C08989=1033.832,386.586,-137.871,173.247,46.071,159.158
C08990=1033.841,386.832,-137.913,173.256,46.074,159.159
C08991=1033.850,387.077,-137.956,173.264,46.078,159.161
C08992=1033.859,387.324,-137.998,173.272,46.082,159.163
C08993=1033.868,387.571,-138.041,173.280,46.085,159.165
C08994=1033.878,387.816,-138.083,173.289,46.089,159.167
C08995=1033.886,388.062,-138.126,173.297,46.092,159.169
C08996=1033.895,388.309,-138.168,173.306,46.096,159.171
C08997=1033.904,388.554,-138.210,173.314,46.100,159.173
C08998=1033.913,388.801,-138.254,173.324,46.103,159.175
C08999=1033.923,389.047,-138.296,173.332,46.106,159.176
C09000=1033.931,389.293,-138.339,173.341,46.110,159.178
C09001=1033.941,389.539,-138.382,173.350,46.114,159.180
C09002=1033.950,389.785,-138.424,173.358,46.117,159.182
C09003=1033.959,390.031,-138.467,173.367,46.121,159.184
C09004=1033.969,390.278,-138.510,173.376,46.125,159.186
C09005=1033.977,390.524,-138.553,173.384,46.129,159.188
C09006=1033.987,390.770,-138.597,173.393,46.132,159.190
C09007=1033.996,391.016,-138.640,173.402,46.136,159.192
C09008=1034.005,391.261,-138.682,173.410,46.140,159.194
C09009=1034.014,391.508,-138.726,173.420,46.143,159.196
C09010=1034.024,391.753,-138.769,173.429,46.147,159.198
C09011=1034.033,392.000,-138.812,173.437,46.151,159.200
C09012=1034.042,392.246,-138.855,173.446,46.155,159.202
C09013=1034.051,392.492,-138.899,173.455,46.159,159.204
C09014=1034.060,392.726,-138.940,173.463,46.162,159.206
C09015=1034.069,392.960,-138.981,173.472,46.166,159.208
C09016=1034.078,393.195,-139.022,173.481,46.170,159.210
C09017=1034.087,393.430,-139.063,173.489,46.173,159.212
C09018=1034.096,393.664,-139.105,173.498,46.177,159.214
C09019=1034.105,393.898,-139.146,173.507,46.181,159.216
C09020=1034.114,394.134,-139.188,173.515,46.184,159.218
C09021=1034.123,394.368,-139.229,173.524,46.188,159.220
C09022=1034.132,394.614,-139.273,173.533,46.192,159.222
C09023=1034.141,394.860,-139.317,173.542,46.196,159.224
C09024=1034.151,395.105,-139.360,173.551,46.200,159.226
C09025=1034.160,395.352,-139.404,173.560,46.204,159.228
C09026=1034.170,395.598,-139.448,173.570,46.208,159.230
C09027=1034.179,395.843,-139.491,173.579,46.212,159.232
C09028=1034.188,396.089,-139.535,173.588,46.216,159.234
C09029=1034.198,396.335,-139.579,173.598,46.220,159.237
C09030=1034.207,396.582,-139.623,173.607,46.224,159.239
C09031=1034.217,396.827,-139.667,173.617,46.228,159.241
C09032=1034.227,397.072,-139.711,173.626,46.233,159.243
C09033=1034.236,397.318,-139.755,173.635,46.237,159.245
C09034=1034.245,397.565,-139.799,173.645,46.241,159.247
C09035=1034.256,397.810,-139.843,173.654,46.245,159.250
C09036=1034.265,398.056,-139.887,173.664,46.249,159.252
C09037=1034.275,398.302,-139.932,173.673,46.253,159.254
C09038=1034.284,398.548,-139.976,173.683,46.257,159.256
C09039=1034.294,398.794,-140.019,173.692,46.261,159.258
C09040=1034.304,399.039,-140.064,173.701,46.265,159.260
C09041=1034.313,399.286,-140.108,173.712,46.270,159.263
C09042=1034.323,399.532,-140.152,173.721,46.274,159.265
C09043=1034.332,399.777,-140.197,173.731,46.278,159.267
C09044=1034.343,400.022,-140.241,173.740,46.283,159.270
C09045=1034.352,400.269,-140.286,173.750,46.287,159.272
C09046=1034.362,400.514,-140.330,173.759,46.292,159.274
C09047=1034.371,400.760,-140.375,173.769,46.296,159.276
C09048=1034.381,401.006,-140.419,173.779,46.300,159.279
C09049=1034.391,401.251,-140.464,173.788,46.304,159.281
C09050=1034.401,401.497,-140.509,173.799,46.309,159.283
C09051=1034.410,401.742,-140.554,173.809,46.313,159.286
C09052=1034.420,401.989,-140.598,173.818,46.317,159.288
C09053=1034.430,402.235,-140.643,173.828,46.322,159.290
C09054=1034.440,402.480,-140.688,173.838,46.326,159.293
C09055=1034.449,402.726,-140.733,173.848,46.331,159.295
C09056=1034.460,402.972,-140.778,173.858,46.336,159.297
C09057=1034.470,403.217,-140.823,173.868,46.340,159.300
C09058=1034.478,403.463,-140.868,173.879,46.345,159.302
C09059=1034.489,403.708,-140.914,173.888,46.349,159.305
C09060=1034.499,403.954,-140.959,173.898,46.354,159.307
C09061=1034.509,404.200,-141.004,173.908,46.358,159.309
C09062=1034.518,404.445,-141.049,173.919,46.363,159.312
C09063=1034.529,404.691,-141.094,173.929,46.367,159.314
C09064=1034.538,404.937,-141.140,173.939,46.372,159.317
C09065=1034.548,405.183,-141.185,173.949,46.377,159.319
C09066=1034.558,405.428,-141.231,173.959,46.382,159.322
C09067=1034.569,405.674,-141.276,173.970,46.386,159.324
C09068=1034.579,405.919,-141.321,173.980,46.390,159.326
C09069=1034.588,406.166,-141.367,173.990,46.396,159.329
C09070=1034.598,406.403,-141.412,174.001,46.400,159.331
C09071=1034.608,406.640,-141.455,174.010,46.405,159.334
C09072=1034.618,406.877,-141.499,174.020,46.409,159.336
C09073=1034.627,407.114,-141.543,174.031,46.414,159.339
C09074=1034.637,407.355,-141.588,174.041,46.419,159.341
C09075=1034.647,407.596,-141.633,174.052,46.423,159.344
C09076=1034.658,407.837,-141.678,174.062,46.427,159.346
C09077=1034.667,408.077,-141.722,174.071,46.433,159.349
C09078=1034.677,408.318,-141.767,174.082,46.437,159.351
C09079=1034.688,408.558,-141.813,174.092,46.442,159.354
C09080=1034.698,408.799,-141.857,174.103,46.447,159.356
C09081=1034.707,409.040,-141.903,174.113,46.452,159.359
C09082=1034.718,409.286,-141.949,174.124,46.457,159.361
C09083=1034.728,409.531,-141.994,174.135,46.461,159.364
C09084=1034.739,409.776,-142.040,174.146,46.466,159.367
C09085=1034.749,410.022,-142.086,174.157,46.471,159.369
C09086=1034.760,410.267,-142.133,174.167,46.476,159.372
C09087=1034.770,410.513,-142.179,174.178,46.481,159.374
C09088=1034.781,410.758,-142.225,174.190,46.486,159.377
C09089=1034.791,411.004,-142.271,174.201,46.491,159.380
C09090=1034.802,411.249,-142.318,174.211,46.496,159.382
C09091=1034.812,411.495,-142.364,174.222,46.501,159.385
C09092=1034.822,411.740,-142.411,174.234,46.507,159.388
C09093=1034.833,411.986,-142.457,174.244,46.512,159.391
C09094=1034.843,412.231,-142.504,174.255,46.517,159.393
C09095=1034.854,412.477,-142.550,174.267,46.522,159.396
C09096=1034.864,412.722,-142.597,174.278,46.527,159.399
C09097=1034.874,412.967,-142.645,174.289,46.533,159.402
C09098=1034.885,413.213,-142.691,174.300,46.537,159.404
C09099=1034.895,413.458,-142.738,174.311,46.543,159.407
C09100=1034.906,413.703,-142.784,174.323,46.548,159.410
C09101=1034.917,413.949,-142.832,174.334,46.554,159.413
C09102=1034.928,414.194,-142.879,174.346,46.558,159.416
C09103=1034.938,414.439,-142.926,174.357,46.564,159.418
C09104=1034.949,414.684,-142.972,174.369,46.569,159.421
C09105=1034.959,414.930,-143.020,174.380,46.574,159.424
C09106=1034.970,415.176,-143.067,174.392,46.580,159.427
C09107=1034.981,415.420,-143.114,174.403,46.585,159.430
C09108=1034.991,415.666,-143.161,174.415,46.591,159.433
C09109=1035.002,415.911,-143.208,174.426,46.596,159.436
C09110=1035.013,416.157,-143.255,174.438,46.602,159.439
C09111=1035.025,416.402,-143.303,174.450,46.607,159.441
C09112=1035.035,416.647,-143.350,174.461,46.613,159.444
C09113=1035.046,416.893,-143.397,174.473,46.618,159.447
C09114=1035.057,417.137,-143.445,174.485,46.623,159.450
C09115=1035.068,417.383,-143.493,174.497,46.629,159.453
C09116=1035.078,417.628,-143.541,174.509,46.635,159.456
C09117=1035.090,417.874,-143.588,174.521,46.640,159.459
C09118=1035.100,418.118,-143.636,174.533,46.646,159.462
C09119=1035.111,418.364,-143.684,174.545,46.651,159.465
C09120=1035.121,418.609,-143.731,174.556,46.657,159.468
C09121=1035.132,418.854,-143.779,174.568,46.663,159.471
C09122=1035.144,419.100,-143.828,174.581,46.668,159.474
C09123=1035.155,419.344,-143.875,174.593,46.674,159.477
C09124=1035.166,419.589,-143.923,174.605,46.680,159.480
C09125=1035.177,419.835,-143.972,174.618,46.685,159.484
C09126=1035.187,420.079,-144.020,174.630,46.691,159.487
C09127=1035.199,420.325,-144.068,174.642,46.697,159.490
C09128=1035.210,420.570,-144.116,174.655,46.703,159.493
C09129=1035.222,420.815,-144.164,174.667,46.709,159.496
C09130=1035.233,421.061,-144.212,174.679,46.714,159.499
C09131=1035.243,421.305,-144.260,174.692,46.720,159.502
C09132=1035.255,421.550,-144.309,174.704,46.726,159.506
C09133=1035.266,421.795,-144.357,174.717,46.732,159.509
C09134=1035.277,422.041,-144.406,174.729,46.738,159.512
C09135=1035.288,422.286,-144.455,174.742,46.744,159.515
C09136=1035.300,422.531,-144.502,174.754,46.750,159.518
C09137=1035.311,422.775,-144.551,174.767,46.756,159.522
C09138=1035.323,423.021,-144.600,174.780,46.762,159.525
C09139=1035.334,423.266,-144.649,174.793,46.768,159.528
C09140=1035.346,423.511,-144.697,174.805,46.774,159.531
C09141=1035.357,423.756,-144.746,174.818,46.780,159.535
C09142=1035.368,424.001,-144.795,174.832,46.786,159.538
C09143=1035.380,424.246,-144.844,174.844,46.792,159.541
C09144=1035.391,424.490,-144.893,174.857,46.798,159.545
C09145=1035.403,424.735,-144.942,174.871,46.804,159.548
C09146=1035.414,424.982,-144.992,174.883,46.810,159.551
C09147=1035.425,425.226,-145.041,174.896,46.817,159.555
C09148=1035.437,425.470,-145.090,174.910,46.823,159.558
C09149=1035.448,425.715,-145.139,174.923,46.829,159.561
C09150=1035.460,425.961,-145.189,174.936,46.835,159.565
C09151=1035.471,426.205,-145.238,174.949,46.842,159.568
C09152=1035.483,426.450,-145.287,174.963,46.848,159.572
C09153=1035.495,426.695,-145.337,174.976,46.854,159.575
C09154=1035.507,426.940,-145.386,174.990,46.861,159.579
C09155=1035.519,427.185,-145.435,175.003,46.867,159.582
C09156=1035.530,427.429,-145.485,175.016,46.873,159.585
C09157=1035.542,427.675,-145.535,175.030,46.879,159.589
C09158=1035.553,427.919,-145.585,175.043,46.886,159.593
C09159=1035.566,428.164,-145.635,175.057,46.892,159.596
C09160=1035.577,428.408,-145.685,175.071,46.899,159.600
C09161=1035.589,428.654,-145.735,175.084,46.905,159.603
C09162=1035.600,428.898,-145.784,175.099,46.912,159.607
C09163=1035.612,429.143,-145.835,175.113,46.919,159.610
C09164=1035.624,429.387,-145.885,175.127,46.925,159.614
C09165=1035.636,429.632,-145.935,175.141,46.931,159.618
C09166=1035.647,429.877,-145.986,175.154,46.939,159.621
C09167=1035.659,430.121,-146.035,175.168,46.945,159.625
C09168=1035.672,430.366,-146.085,175.182,46.952,159.629
C09169=1035.683,430.611,-146.137,175.196,46.958,159.632
C09170=1035.696,430.855,-146.187,175.211,46.965,159.636
C09171=1035.708,431.100,-146.237,175.225,46.972,159.640
C09172=1035.719,431.345,-146.287,175.239,46.979,159.644
C09173=1035.732,431.589,-146.338,175.254,46.985,159.647
C09174=1035.744,431.834,-146.388,175.268,46.992,159.651
C09175=1035.757,432.078,-146.439,175.282,46.999,159.655
C09176=1035.768,432.323,-146.490,175.297,47.005,159.659
C09177=1035.781,432.567,-146.541,175.312,47.012,159.663
C09178=1035.793,432.811,-146.591,175.326,47.019,159.666
C09179=1035.805,433.057,-146.642,175.341,47.026,159.670
C09180=1035.818,433.301,-146.693,175.355,47.033,159.674
C09181=1035.830,433.545,-146.744,175.371,47.040,159.678
C09182=1035.842,433.789,-146.795,175.385,47.047,159.682
C09183=1035.855,434.034,-146.846,175.400,47.054,159.686
C09184=1035.867,434.279,-146.898,175.415,47.060,159.690
C09185=1035.880,434.523,-146.948,175.430,47.068,159.694
C09186=1035.893,434.768,-147.000,175.445,47.074,159.697
C09187=1035.905,435.013,-147.051,175.460,47.082,159.701
C09188=1035.917,435.257,-147.102,175.475,47.089,159.705
C09189=1035.930,435.501,-147.154,175.490,47.096,159.709
C09190=1035.942,435.746,-147.206,175.505,47.103,159.713
C09191=1035.955,435.990,-147.257,175.521,47.110,159.717
C09192=1035.967,436.234,-147.309,175.537,47.117,159.721
C09193=1035.980,436.479,-147.360,175.552,47.125,159.726
C09194=1035.993,436.725,-147.412,175.567,47.132,159.730
C09195=1036.006,436.971,-147.465,175.583,47.139,159.734
C09196=1036.018,437.216,-147.516,175.598,47.147,159.738
C09197=1036.031,437.462,-147.569,175.614,47.154,159.742
C09198=1036.044,437.707,-147.621,175.630,47.161,159.746
C09199=1036.057,437.951,-147.674,175.646,47.169,159.751
C09200=1036.070,438.195,-147.725,175.662,47.176,159.755
C09201=1036.082,438.440,-147.778,175.677,47.184,159.759
C09202=1036.095,438.683,-147.830,175.693,47.191,159.763
C09203=1036.108,438.928,-147.882,175.709,47.198,159.767
C09204=1036.121,439.172,-147.934,175.725,47.206,159.772
C09205=1036.134,439.417,-147.987,175.741,47.214,159.776
C09206=1036.147,439.660,-148.039,175.757,47.221,159.780
C09207=1036.160,439.904,-148.091,175.773,47.228,159.785
C09208=1036.173,440.148,-148.145,175.789,47.236,159.789
C09209=1036.186,440.393,-148.196,175.807,47.243,159.793
C09210=1036.199,440.637,-148.250,175.823,47.251,159.798
C09211=1036.212,440.881,-148.302,175.839,47.259,159.802
C09212=1036.225,441.125,-148.355,175.856,47.267,159.807
C09213=1036.238,441.369,-148.408,175.872,47.274,159.811
C09214=1036.252,441.613,-148.461,175.889,47.282,159.816
C09215=1036.265,441.857,-148.514,175.906,47.290,159.820
C09216=1036.278,442.101,-148.568,175.922,47.297,159.825
C09217=1036.292,442.345,-148.621,175.940,47.305,159.829
C09218=1036.305,442.588,-148.673,175.956,47.313,159.834
C09219=1036.319,442.832,-148.727,175.973,47.320,159.838
C09220=1036.332,443.076,-148.780,175.990,47.329,159.843
C09221=1036.345,443.320,-148.833,176.008,47.336,159.847
C09222=1036.359,443.563,-148.886,176.024,47.344,159.852
C09223=1036.372,443.807,-148.939,176.042,47.352,159.857
C09224=1036.386,444.050,-148.993,176.058,47.360,159.861
C09225=1036.399,444.294,-149.046,176.076,47.368,159.866
C09226=1036.414,444.537,-149.099,176.094,47.376,159.870
C09227=1036.429,444.780,-149.150,176.111,47.384,159.875
C09228=1036.445,445.024,-149.203,176.129,47.391,159.880
C09229=1036.461,445.267,-149.254,176.146,47.399,159.884
C09230=1036.478,445.511,-149.305,176.164,47.406,159.889
C09231=1036.495,445.755,-149.355,176.182,47.413,159.893
C09232=1036.513,445.999,-149.405,176.200,47.421,159.898
C09233=1036.531,446.243,-149.455,176.218,47.428,159.903
C09234=1036.550,446.486,-149.503,176.236,47.435,159.907
C09235=1036.569,446.731,-149.553,176.254,47.442,159.911
C09236=1036.589,446.975,-149.601,176.272,47.449,159.916
C09237=1036.609,447.220,-149.649,176.291,47.456,159.921
C09238=1036.630,447.464,-149.696,176.309,47.462,159.925
C09239=1036.652,447.708,-149.743,176.327,47.469,159.929
C09240=1036.673,447.953,-149.789,176.346,47.475,159.934
C09241=1036.697,448.198,-149.835,176.364,47.482,159.938
C09242=1036.719,448.442,-149.881,176.383,47.488,159.943
C09243=1036.743,448.687,-149.926,176.401,47.495,159.947
C09244=1036.767,448.931,-149.971,176.421,47.501,159.952
C09245=1036.792,449.177,-150.015,176.440,47.507,159.956
C09246=1036.817,449.422,-150.059,176.459,47.513,159.961
C09247=1036.843,449.667,-150.102,176.478,47.519,159.965
C09248=1036.869,449.912,-150.145,176.497,47.525,159.969
C09249=1036.896,450.157,-150.188,176.517,47.530,159.974
C09250=1036.924,450.403,-150.229,176.536,47.536,159.978
C09251=1036.951,450.649,-150.271,176.555,47.541,159.982
C09252=1036.980,450.893,-150.313,176.575,47.548,159.987
C09253=1037.009,451.139,-150.353,176.594,47.553,159.991
C09254=1037.046,451.441,-150.403,176.619,47.560,159.996
C09255=1037.083,451.744,-150.451,176.644,47.566,160.002
C09256=1037.122,452.046,-150.499,176.668,47.572,160.007
C09257=1037.160,452.347,-150.547,176.693,47.578,160.012
C09258=1036.869,452.403,-150.871,176.696,47.649,160.034
C09259=1036.832,452.115,-150.826,176.672,47.644,160.029
C09260=1036.796,451.826,-150.779,176.648,47.637,160.024
C09261=1036.760,451.537,-150.733,176.625,47.632,160.019
C09262=1036.724,451.248,-150.686,176.602,47.626,160.014
C09263=1036.695,451.003,-150.646,176.582,47.620,160.010
C09264=1036.666,450.758,-150.605,176.562,47.615,160.006
C09265=1036.638,450.512,-150.564,176.543,47.609,160.001
C09266=1036.610,450.266,-150.522,176.523,47.604,159.997
C09267=1036.583,450.021,-150.480,176.504,47.598,159.992
C09268=1036.557,449.776,-150.437,176.484,47.592,159.988
C09269=1036.531,449.531,-150.394,176.465,47.586,159.984
C09270=1036.504,449.286,-150.350,176.446,47.580,159.979
C09271=1036.480,449.041,-150.307,176.427,47.574,159.975
C09272=1036.455,448.796,-150.261,176.408,47.569,159.971
C09273=1036.431,448.551,-150.217,176.389,47.562,159.966
C09274=1036.407,448.306,-150.171,176.371,47.556,159.962
C09275=1036.385,448.062,-150.126,176.351,47.549,159.957
C09276=1036.363,447.816,-150.080,176.333,47.543,159.953
C09277=1036.341,447.572,-150.033,176.314,47.537,159.948
C09278=1036.319,447.328,-149.986,176.296,47.530,159.944
C09279=1036.298,447.084,-149.938,176.278,47.523,159.939
C09280=1036.279,446.839,-149.890,176.259,47.517,159.935
C09281=1036.259,446.595,-149.841,176.241,47.510,159.930
C09282=1036.240,446.351,-149.794,176.223,47.503,159.926
C09283=1036.221,446.107,-149.744,176.204,47.496,159.921
C09284=1036.203,445.863,-149.694,176.187,47.489,159.917
C09285=1036.185,445.619,-149.644,176.168,47.482,159.912
C09286=1036.169,445.375,-149.593,176.151,47.474,159.908
C09287=1036.152,445.132,-149.542,176.133,47.467,159.903
C09288=1036.137,444.888,-149.491,176.116,47.459,159.898
C09289=1036.121,444.645,-149.439,176.098,47.452,159.894
C09290=1036.106,444.402,-149.387,176.081,47.444,159.889
C09291=1036.092,444.159,-149.333,176.063,47.437,159.885
C09292=1036.078,443.915,-149.281,176.046,47.429,159.880
C09293=1036.065,443.672,-149.227,176.029,47.421,159.875
C09294=1036.051,443.429,-149.173,176.011,47.413,159.871
C09295=1036.038,443.185,-149.120,175.994,47.405,159.866
C09296=1036.025,442.941,-149.067,175.977,47.398,159.862
C09297=1036.011,442.697,-149.014,175.960,47.390,159.857
C09298=1035.997,442.453,-148.961,175.943,47.382,159.852
C09299=1035.984,442.209,-148.907,175.926,47.375,159.848
C09300=1035.970,441.966,-148.854,175.910,47.367,159.843
C09301=1035.957,441.721,-148.802,175.892,47.359,159.839
C09302=1035.944,441.477,-148.749,175.876,47.351,159.834
C09303=1035.931,441.233,-148.695,175.859,47.344,159.830
C09304=1035.917,440.989,-148.643,175.842,47.336,159.825
C09305=1035.904,440.745,-148.590,175.826,47.328,159.821
C09306=1035.891,440.501,-148.537,175.809,47.321,159.817
C09307=1035.878,440.257,-148.484,175.793,47.314,159.812
C09308=1035.866,440.013,-148.432,175.777,47.306,159.808
C09309=1035.852,439.769,-148.379,175.761,47.298,159.804
C09310=1035.839,439.525,-148.327,175.744,47.291,159.799
C09311=1035.826,439.281,-148.273,175.728,47.284,159.795
C09312=1035.813,439.036,-148.222,175.711,47.276,159.791
C09313=1035.800,438.793,-148.169,175.695,47.269,159.786
C09314=1035.787,438.548,-148.118,175.679,47.262,159.782
C09315=1035.774,438.304,-148.065,175.664,47.255,159.778
C09316=1035.762,438.060,-148.013,175.648,47.247,159.774
C09317=1035.748,437.815,-147.961,175.632,47.239,159.769
C09318=1035.736,437.571,-147.909,175.617,47.233,159.765
C09319=1035.723,437.324,-147.855,175.600,47.225,159.761
C09320=1035.710,437.076,-147.803,175.584,47.218,159.757
C09321=1035.697,436.829,-147.751,175.569,47.211,159.753
C09322=1035.684,436.582,-147.698,175.553,47.203,159.749
C09323=1035.672,436.338,-147.647,175.538,47.196,159.745
C09324=1035.659,436.094,-147.595,175.522,47.189,159.740
C09325=1035.646,435.849,-147.543,175.506,47.182,159.736
C09326=1035.634,435.605,-147.492,175.492,47.175,159.732
C09327=1035.622,435.361,-147.441,175.476,47.168,159.728
C09328=1035.608,435.116,-147.389,175.461,47.161,159.724
C09329=1035.596,434.872,-147.337,175.446,47.154,159.720
C09330=1035.584,434.628,-147.286,175.431,47.147,159.716
C09331=1035.572,434.383,-147.235,175.415,47.140,159.712
C09332=1035.559,434.138,-147.184,175.401,47.133,159.709
C09333=1035.547,433.894,-147.132,175.387,47.126,159.705
C09334=1035.534,433.650,-147.082,175.371,47.119,159.701
C09335=1035.522,433.405,-147.032,175.356,47.112,159.697
C09336=1035.510,433.160,-146.980,175.341,47.106,159.693
C09337=1035.497,432.915,-146.929,175.326,47.099,159.689
C09338=1035.484,432.671,-146.878,175.312,47.092,159.685
C09339=1035.472,432.426,-146.827,175.298,47.085,159.681
C09340=1035.460,432.182,-146.777,175.283,47.078,159.678
C09341=1035.447,431.938,-146.726,175.268,47.072,159.674
C09342=1035.435,431.694,-146.676,175.254,47.065,159.670
C09343=1035.424,431.448,-146.625,175.239,47.059,159.666
C09344=1035.411,431.204,-146.575,175.225,47.052,159.663
C09345=1035.399,430.959,-146.524,175.211,47.045,159.659
C09346=1035.387,430.714,-146.474,175.197,47.039,159.655
C09347=1035.375,430.470,-146.423,175.182,47.032,159.651
C09348=1035.363,430.226,-146.373,175.168,47.025,159.648
C09349=1035.351,429.981,-146.323,175.154,47.019,159.644
C09350=1035.339,429.736,-146.272,175.140,47.012,159.641
C09351=1035.327,429.491,-146.222,175.126,47.006,159.637
C09352=1035.316,429.247,-146.172,175.112,47.000,159.633
C09353=1035.304,429.002,-146.122,175.098,46.992,159.630
C09354=1035.292,428.758,-146.072,175.084,46.986,159.626
C09355=1035.280,428.513,-146.022,175.070,46.980,159.622
C09356=1035.269,428.268,-145.972,175.056,46.973,159.619
C09357=1035.257,428.023,-145.922,175.042,46.967,159.615
C09358=1035.245,427.779,-145.873,175.029,46.960,159.612
C09359=1035.233,427.534,-145.822,175.016,46.955,159.608
C09360=1035.222,427.289,-145.773,175.002,46.948,159.605
C09361=1035.210,427.044,-145.723,174.989,46.942,159.601
C09362=1035.198,426.799,-145.674,174.975,46.936,159.598
C09363=1035.186,426.554,-145.625,174.961,46.929,159.594
C09364=1035.174,426.310,-145.575,174.948,46.923,159.591
C09365=1035.162,426.064,-145.525,174.934,46.917,159.587
C09366=1035.151,425.820,-145.476,174.921,46.911,159.584
C09367=1035.140,425.575,-145.427,174.907,46.904,159.581
C09368=1035.128,425.329,-145.377,174.895,46.898,159.577
C09369=1035.117,425.085,-145.328,174.881,46.892,159.574
C09370=1035.105,424.840,-145.279,174.868,46.886,159.571
C09371=1035.094,424.596,-145.230,174.856,46.880,159.567
C09372=1035.083,424.350,-145.181,174.842,46.874,159.564
C09373=1035.071,424.105,-145.132,174.829,46.868,159.561
C09374=1035.059,423.860,-145.083,174.816,46.862,159.557
C09375=1035.048,423.615,-145.034,174.803,46.856,159.554
C09376=1035.037,423.371,-144.985,174.790,46.850,159.551
C09377=1035.025,423.125,-144.937,174.778,46.844,159.548
C09378=1035.014,422.880,-144.888,174.764,46.838,159.544
C09379=1035.003,422.633,-144.839,174.752,46.832,159.541
C09380=1034.990,422.386,-144.790,174.739,46.826,159.538
C09381=1034.979,422.138,-144.741,174.726,46.821,159.534
C09382=1034.968,421.890,-144.692,174.713,46.814,159.531
C09383=1034.957,421.645,-144.644,174.701,46.809,159.528
C09384=1034.945,421.400,-144.595,174.688,46.803,159.525
C09385=1034.934,421.155,-144.547,174.676,46.797,159.522
C09386=1034.923,420.910,-144.499,174.663,46.791,159.519
C09387=1034.912,420.665,-144.451,174.651,46.786,159.515
C09388=1034.901,420.421,-144.402,174.639,46.780,159.512
C09389=1034.890,420.175,-144.353,174.626,46.774,159.509
C09390=1034.878,419.930,-144.305,174.614,46.769,159.506
C09391=1034.867,419.685,-144.258,174.602,46.763,159.503
C09392=1034.856,419.440,-144.209,174.590,46.757,159.500
C09393=1034.845,419.194,-144.162,174.577,46.752,159.497
C09394=1034.834,418.949,-144.113,174.565,46.746,159.494
C09395=1034.824,418.704,-144.066,174.553,46.740,159.491
C09396=1034.813,418.459,-144.017,174.541,46.735,159.488
C09397=1034.801,418.214,-143.970,174.528,46.729,159.485
C09398=1034.791,417.968,-143.922,174.517,46.723,159.482
C09399=1034.780,417.724,-143.874,174.505,46.718,159.479
C09400=1034.769,417.478,-143.826,174.493,46.712,159.476
C09401=1034.759,417.233,-143.779,174.481,46.707,159.473
C09402=1034.747,416.988,-143.731,174.468,46.702,159.470
C09403=1034.737,416.743,-143.684,174.457,46.696,159.467
C09404=1034.725,416.497,-143.637,174.445,46.691,159.464
C09405=1034.715,416.252,-143.589,174.433,46.686,159.461
C09406=1034.703,416.007,-143.542,174.422,46.680,159.458
C09407=1034.693,415.761,-143.495,174.410,46.675,159.455
C09408=1034.682,415.515,-143.447,174.398,46.669,159.452
C09409=1034.671,415.271,-143.401,174.387,46.664,159.449
C09410=1034.661,415.025,-143.353,174.375,46.659,159.446
C09411=1034.650,414.780,-143.306,174.363,46.654,159.444
C09412=1034.639,414.535,-143.259,174.352,46.648,159.441
C09413=1034.628,414.289,-143.213,174.340,46.643,159.438
C09414=1034.618,414.044,-143.165,174.330,46.638,159.435
C09415=1034.607,413.799,-143.119,174.318,46.633,159.432
C09416=1034.597,413.553,-143.071,174.307,46.627,159.430
C09417=1034.586,413.308,-143.025,174.295,46.623,159.427
C09418=1034.575,413.063,-142.977,174.284,46.617,159.424
C09419=1034.566,412.817,-142.931,174.272,46.612,159.421
C09420=1034.555,412.572,-142.884,174.261,46.607,159.419
C09421=1034.544,412.327,-142.837,174.250,46.602,159.416
C09422=1034.534,412.081,-142.791,174.239,46.597,159.413
C09423=1034.524,411.836,-142.744,174.228,46.591,159.410
C09424=1034.513,411.590,-142.698,174.217,46.586,159.408
C09425=1034.503,411.345,-142.651,174.205,46.582,159.405
C09426=1034.492,411.099,-142.605,174.194,46.576,159.402
C09427=1034.482,410.854,-142.558,174.184,46.571,159.399
C09428=1034.471,410.608,-142.512,174.172,46.567,159.397
C09429=1034.461,410.363,-142.466,174.162,46.562,159.394
C09430=1034.450,410.117,-142.420,174.151,46.557,159.391
C09431=1034.440,409.871,-142.373,174.140,46.552,159.389
C09432=1034.430,409.626,-142.328,174.129,46.547,159.386
C09433=1034.419,409.381,-142.281,174.118,46.542,159.384
C09434=1034.408,409.135,-142.235,174.108,46.538,159.381
C09435=1034.398,408.893,-142.190,174.097,46.533,159.378
C09436=1034.389,408.651,-142.145,174.086,46.528,159.376
C09437=1034.378,408.410,-142.100,174.076,46.523,159.373
C09438=1034.367,408.168,-142.054,174.065,46.518,159.371
C09439=1034.358,407.926,-142.010,174.055,46.514,159.368
C09440=1034.347,407.685,-141.964,174.044,46.509,159.366
C09441=1034.338,407.443,-141.919,174.034,46.504,159.363
C09442=1034.328,407.201,-141.874,174.024,46.500,159.361
C09443=1034.317,406.955,-141.828,174.013,46.495,159.358
C09444=1034.308,406.710,-141.784,174.003,46.491,159.356
C09445=1034.297,406.464,-141.738,173.992,46.486,159.353
C09446=1034.287,406.219,-141.692,173.982,46.481,159.351
C09447=1034.277,405.973,-141.646,173.972,46.477,159.348
C09448=1034.267,405.728,-141.601,173.961,46.472,159.346
C09449=1034.257,405.482,-141.556,173.951,46.467,159.343
C09450=1034.247,405.237,-141.510,173.940,46.463,159.341
C09451=1034.237,404.991,-141.465,173.930,46.458,159.339
C09452=1034.228,404.745,-141.419,173.920,46.454,159.336
C09453=1034.217,404.499,-141.374,173.909,46.449,159.333
C09454=1034.207,404.254,-141.329,173.900,46.444,159.331
C09455=1034.198,404.008,-141.284,173.889,46.440,159.329
C09456=1034.187,403.763,-141.238,173.879,46.435,159.326
C09457=1034.177,403.517,-141.193,173.869,46.431,159.324
C09458=1034.168,403.271,-141.148,173.859,46.427,159.322
C09459=1034.158,403.025,-141.103,173.850,46.422,159.319
C09460=1034.148,402.779,-141.058,173.839,46.418,159.317
C09461=1034.139,402.534,-141.013,173.829,46.413,159.314
C09462=1034.129,402.288,-140.968,173.819,46.409,159.312
C09463=1034.118,402.042,-140.923,173.809,46.405,159.310
C09464=1034.109,401.797,-140.878,173.799,46.400,159.307
C09465=1034.099,401.551,-140.833,173.789,46.395,159.305
C09466=1034.089,401.306,-140.788,173.779,46.391,159.303
C09467=1034.080,401.060,-140.744,173.770,46.387,159.300
C09468=1034.070,400.814,-140.699,173.760,46.383,159.298
C09469=1034.060,400.568,-140.654,173.749,46.378,159.296
C09470=1034.050,400.322,-140.610,173.740,46.374,159.294
C09471=1034.040,400.077,-140.566,173.730,46.370,159.291
C09472=1034.030,399.831,-140.521,173.720,46.366,159.289
C09473=1034.021,399.585,-140.477,173.711,46.361,159.287
C09474=1034.011,399.339,-140.432,173.701,46.358,159.285
C09475=1034.002,399.093,-140.388,173.692,46.353,159.282
C09476=1033.992,398.847,-140.344,173.682,46.349,159.280
C09477=1033.982,398.602,-140.300,173.672,46.345,159.278
C09478=1033.973,398.356,-140.256,173.663,46.341,159.276
C09479=1033.963,398.110,-140.212,173.653,46.337,159.273
C09480=1033.953,397.864,-140.167,173.644,46.332,159.271
C09481=1033.944,397.619,-140.124,173.634,46.328,159.269
C09482=1033.934,397.373,-140.079,173.625,46.324,159.267
C09483=1033.925,397.145,-140.038,173.616,46.321,159.265
C09484=1033.917,396.916,-139.998,173.608,46.317,159.263
C09485=1033.908,396.687,-139.956,173.599,46.313,159.261
C09486=1033.899,396.460,-139.916,173.590,46.310,159.259
C09487=1033.890,396.231,-139.876,173.582,46.306,159.257
C09488=1033.881,396.003,-139.834,173.573,46.302,159.255
C09489=1033.873,395.775,-139.793,173.564,46.299,159.253
C09490=1033.863,395.546,-139.754,173.556,46.295,159.251
C09491=1033.854,395.300,-139.709,173.547,46.291,159.249
C09492=1033.845,395.055,-139.666,173.537,46.287,159.247
C09493=1033.836,394.809,-139.622,173.528,46.283,159.245
C09494=1033.826,394.563,-139.578,173.519,46.279,159.243
C09495=1033.817,394.317,-139.535,173.509,46.276,159.241
C09496=1033.808,394.071,-139.491,173.500,46.271,159.238
C09497=1033.798,393.825,-139.447,173.492,46.268,159.236
C09498=1033.789,393.579,-139.404,173.482,46.264,159.234
C09499=1033.779,393.327,-139.359,173.473,46.260,159.232
C09500=1033.769,393.074,-139.315,173.463,46.256,159.230
C09501=1033.760,392.822,-139.271,173.454,46.252,159.228
C09502=1033.750,392.570,-139.226,173.445,46.248,159.226
C09503=1033.741,392.324,-139.183,173.436,46.245,159.224
C09504=1033.732,392.078,-139.140,173.427,46.241,159.222
C09505=1033.722,391.832,-139.097,173.419,46.237,159.220
C09506=1033.713,391.586,-139.053,173.410,46.233,159.218
C09507=1033.704,391.340,-139.011,173.400,46.230,159.216
C09508=1033.695,391.093,-138.967,173.391,46.226,159.214
C09509=1033.685,390.848,-138.924,173.383,46.222,159.212
C09510=1033.677,390.602,-138.881,173.374,46.218,159.210
C09511=1033.667,390.356,-138.838,173.365,46.215,159.208
C09512=1033.658,390.110,-138.795,173.357,46.212,159.206
C09513=1033.648,389.863,-138.753,173.347,46.208,159.204
C09514=1033.639,389.617,-138.710,173.339,46.204,159.202
C09515=1033.631,389.371,-138.667,173.330,46.201,159.200
C09516=1033.621,389.125,-138.624,173.321,46.197,159.198
C09517=1033.612,388.879,-138.581,173.313,46.194,159.197
C09518=1033.603,388.633,-138.539,173.304,46.190,159.195
C09519=1033.594,388.387,-138.496,173.296,46.186,159.193
C09520=1033.585,388.141,-138.453,173.287,46.183,159.191
C09521=1033.575,387.895,-138.411,173.279,46.180,159.189
C09522=1033.567,387.648,-138.369,173.270,46.176,159.187
C09523=1033.558,387.402,-138.326,173.262,46.173,159.185
C09524=1033.548,387.156,-138.283,173.253,46.169,159.183
C09525=1033.539,386.910,-138.241,173.245,46.166,159.181
C09526=1033.530,386.664,-138.199,173.236,46.162,159.179
C09527=1033.521,386.418,-138.156,173.228,46.159,159.178
C09528=1033.512,386.172,-138.115,173.219,46.156,159.176
C09529=1033.503,385.925,-138.071,173.211,46.152,159.174
C09530=1033.494,385.679,-138.030,173.202,46.149,159.172
C09531=1033.485,385.433,-137.987,173.194,46.146,159.170
C09532=1033.476,385.187,-137.945,173.186,46.143,159.169
C09533=1033.467,384.940,-137.904,173.177,46.139,159.167
C09534=1033.457,384.694,-137.861,173.169,46.136,159.165
C09535=1033.449,384.448,-137.820,173.160,46.132,159.163
C09536=1033.440,384.202,-137.778,173.152,46.129,159.161
C09537=1033.431,383.955,-137.736,173.144,46.126,159.160
C09538=1033.421,383.710,-137.694,173.135,46.123,159.158
C09539=1033.412,383.463,-137.652,173.128,46.120,159.156
C09540=1033.404,383.217,-137.610,173.120,46.116,159.154
C09541=1033.395,382.970,-137.568,173.111,46.113,159.153
C09542=1033.386,382.724,-137.526,173.103,46.110,159.151
C09543=1033.377,382.477,-137.485,173.095,46.107,159.149
C09544=1033.369,382.231,-137.443,173.086,46.104,159.147
C09545=1033.360,381.985,-137.401,173.079,46.100,159.146
C09546=1033.351,381.738,-137.359,173.070,46.097,159.144
C09547=1033.342,381.493,-137.318,173.062,46.094,159.142
C09548=1033.333,381.246,-137.276,173.054,46.091,159.140
C09549=1033.324,381.000,-137.235,173.046,46.088,159.139
C09550=1033.316,380.754,-137.193,173.038,46.085,159.137
C09551=1033.307,380.507,-137.151,173.030,46.082,159.135
C09552=1033.298,380.261,-137.109,173.022,46.079,159.134
C09553=1033.289,380.015,-137.068,173.015,46.075,159.132
C09554=1033.281,379.768,-137.027,173.006,46.072,159.130
C09555=1033.274,379.554,-136.991,173.000,46.070,159.129
C09556=1033.266,379.341,-136.955,172.993,46.067,159.127
C09557=1033.259,379.126,-136.918,172.986,46.065,159.126
C09558=1033.251,378.912,-136.883,172.979,46.062,159.124
C09559=1033.244,378.698,-136.847,172.972,46.060,159.123
C09560=1033.236,378.484,-136.811,172.965,46.057,159.122
C09561=1033.229,378.270,-136.774,172.958,46.055,159.120
C09562=1033.221,378.056,-136.739,172.952,46.051,159.119
C09563=1033.213,377.810,-136.698,172.944,46.049,159.117
C09564=1033.204,377.563,-136.657,172.936,46.046,159.115
C09565=1033.196,377.316,-136.616,172.929,46.043,159.114
C09566=1033.187,377.071,-136.575,172.921,46.040,159.112
C09567=1033.178,376.824,-136.534,172.913,46.038,159.111
C09568=1033.169,376.577,-136.493,172.905,46.034,159.109
C09569=1033.161,376.331,-136.452,172.897,46.031,159.107
C09570=1033.152,376.085,-136.411,172.890,46.029,159.106
C09571=1033.144,375.838,-136.371,172.882,46.026,159.104
C09572=1033.135,375.591,-136.330,172.874,46.023,159.103
C09573=1033.126,375.345,-136.290,172.867,46.020,159.101
C09574=1033.118,375.098,-136.249,172.859,46.018,159.100
C09575=1033.110,374.852,-136.208,172.852,46.015,159.098
C09576=1033.101,374.606,-136.166,172.844,46.012,159.097
C09577=1033.092,374.360,-136.126,172.837,46.009,159.095
C09578=1033.083,374.113,-136.085,172.829,46.007,159.094
C09579=1033.075,373.867,-136.044,172.822,46.004,159.092
C09580=1033.066,373.620,-136.004,172.814,46.001,159.090
C09581=1033.058,373.373,-135.964,172.807,45.998,159.089
C09582=1033.050,373.127,-135.924,172.799,45.996,159.087
C09583=1033.041,372.880,-135.883,172.792,45.993,159.086
C09584=1033.033,372.634,-135.842,172.784,45.990,159.084
C09585=1033.024,372.387,-135.801,172.777,45.987,159.083
C09586=1033.016,372.140,-135.761,172.769,45.985,159.081
C09587=1033.008,371.894,-135.722,172.762,45.982,159.080
C09588=1032.999,371.647,-135.681,172.755,45.979,159.078
C09589=1032.991,371.401,-135.640,172.747,45.977,159.077
C09590=1032.982,371.155,-135.600,172.740,45.974,159.075
C09591=1032.974,370.908,-135.560,172.732,45.972,159.074
C09592=1032.966,370.661,-135.519,172.725,45.969,159.072
C09593=1032.958,370.414,-135.478,172.718,45.967,159.071
C09594=1032.949,370.168,-135.439,172.710,45.964,159.069
C09595=1032.941,369.922,-135.398,172.704,45.962,159.068
C09596=1032.934,369.675,-135.358,172.697,45.959,159.067
C09597=1032.924,369.428,-135.318,172.689,45.957,159.065
C09598=1032.916,369.181,-135.278,172.682,45.954,159.064
C09599=1032.908,368.935,-135.239,172.675,45.951,159.062
C09600=1032.899,368.689,-135.199,172.667,45.949,159.061
C09601=1032.892,368.442,-135.159,172.660,45.946,159.059
C09602=1032.882,368.194,-135.119,172.654,45.944,159.058
C09603=1032.874,367.948,-135.080,172.646,45.942,159.057
C09604=1032.866,367.701,-135.039,172.639,45.939,159.055
C09605=1032.858,367.455,-135.000,172.632,45.937,159.054
C09606=1032.849,367.208,-134.961,172.624,45.935,159.052
C09607=1032.841,366.961,-134.921,172.618,45.932,159.051
C09608=1032.833,366.715,-134.881,172.611,45.929,159.050
C09609=1032.825,366.468,-134.841,172.604,45.927,159.048
C09610=1032.817,366.221,-134.802,172.596,45.925,159.047
C09611=1032.808,365.975,-134.762,172.590,45.923,159.046
C09612=1032.800,365.728,-134.722,172.583,45.920,159.044
C09613=1032.792,365.482,-134.683,172.576,45.918,159.043
C09614=1032.784,365.235,-134.644,172.568,45.916,159.041
C09615=1032.770,364.828,-134.578,172.557,45.912,159.039
C09616=1032.756,364.420,-134.513,172.546,45.908,159.037
C09617=1032.743,364.013,-134.448,172.535,45.904,159.035
C09618=1032.730,363.606,-134.383,172.523,45.900,159.033
C09619=1032.722,363.359,-134.344,172.516,45.898,159.031
C09620=1032.713,363.113,-134.305,172.510,45.896,159.030
C09621=1032.706,362.865,-134.265,172.503,45.894,159.029
C09622=1032.697,362.618,-134.226,172.496,45.892,159.027
C09623=1032.690,362.373,-134.187,172.488,45.890,159.026
C09624=1032.682,362.125,-134.148,172.482,45.887,159.025
C09625=1032.674,361.878,-134.109,172.475,45.885,159.023
C09626=1032.665,361.632,-134.069,172.469,45.883,159.022
C09627=1032.658,361.384,-134.030,172.462,45.881,159.021
C09628=1032.650,361.138,-133.991,172.455,45.878,159.020
C09629=1032.642,360.891,-133.952,172.449,45.877,159.018
C09630=1032.633,360.645,-133.913,172.442,45.874,159.017
C09631=1032.625,360.397,-133.875,172.435,45.872,159.016
C09632=1032.618,360.151,-133.836,172.429,45.870,159.015
C09633=1032.609,359.904,-133.797,172.422,45.868,159.013
C09634=1032.601,359.657,-133.758,172.415,45.866,159.012
C09635=1032.594,359.410,-133.719,172.408,45.864,159.011
C09636=1032.586,359.164,-133.680,172.401,45.862,159.010
C09637=1032.578,358.916,-133.642,172.395,45.860,159.008
C09638=1032.569,358.669,-133.603,172.388,45.858,159.007
C09639=1032.562,358.423,-133.565,172.382,45.856,159.006
C09640=1032.553,358.176,-133.525,172.375,45.854,159.005
C09641=1032.545,357.929,-133.487,172.369,45.852,159.004
C09642=1032.538,357.682,-133.449,172.362,45.850,159.002
C09643=1032.530,357.435,-133.410,172.356,45.848,159.001
C09644=1032.521,357.188,-133.371,172.349,45.846,159.000
C09645=1032.514,356.941,-133.333,172.342,45.844,158.999
C09646=1032.506,356.694,-133.294,172.336,45.842,158.997
C09647=1032.498,356.448,-133.256,172.329,45.840,158.996
C09648=1032.490,356.200,-133.218,172.323,45.839,158.995
C09649=1032.483,355.954,-133.179,172.316,45.836,158.994
C09650=1032.474,355.707,-133.141,172.310,45.834,158.993
C09651=1032.466,355.460,-133.102,172.303,45.833,158.992
C09652=1032.459,355.213,-133.064,172.297,45.831,158.990
C09653=1032.450,354.965,-133.027,172.292,45.829,158.989
C09654=1032.443,354.719,-132.988,172.285,45.827,158.988
C09655=1032.434,354.472,-132.950,172.279,45.825,158.987
C09656=1032.427,354.225,-132.912,172.272,45.824,158.986
C09657=1032.419,353.977,-132.874,172.266,45.822,158.985
C09658=1032.411,353.731,-132.836,172.259,45.820,158.984
C09659=1032.403,353.484,-132.797,172.253,45.818,158.982
C09660=1032.395,353.237,-132.760,172.247,45.816,158.981
C09661=1032.388,352.990,-132.722,172.240,45.815,158.980
C09662=1032.380,352.743,-132.683,172.234,45.813,158.979
C09663=1032.372,352.496,-132.646,172.227,45.811,158.978
C09664=1032.363,352.249,-132.607,172.222,45.809,158.977
C09665=1032.356,352.002,-132.570,172.215,45.807,158.976
C09666=1032.349,351.755,-132.532,172.209,45.806,158.974
C09667=1032.341,351.508,-132.494,172.203,45.804,158.973
C09668=1032.333,351.261,-132.456,172.196,45.803,158.972
C09669=1032.325,351.014,-132.419,172.190,45.801,158.971
C09670=1032.317,350.767,-132.380,172.185,45.799,158.970
C09671=1032.305,350.366,-132.319,172.174,45.796,158.968
C09672=1032.293,349.965,-132.258,172.164,45.794,158.967
C09673=1032.279,349.564,-132.197,172.154,45.791,158.965
C09674=1032.267,349.163,-132.135,172.144,45.788,158.963
C09675=1032.260,348.916,-132.098,172.138,45.786,158.962
C09676=1032.253,348.669,-132.060,172.132,45.785,158.961
C09677=1032.244,348.422,-132.022,172.126,45.783,158.960
C09678=1032.237,348.175,-131.985,172.119,45.782,158.959
C09679=1032.229,347.928,-131.948,172.113,45.780,158.958
C09680=1032.221,347.681,-131.910,172.108,45.778,158.957
C09681=1032.213,347.434,-131.873,172.102,45.777,158.956
C09682=1032.206,347.186,-131.836,172.095,45.775,158.955
C09683=1032.198,346.940,-131.799,172.089,45.774,158.954
C09684=1032.190,346.692,-131.761,172.084,45.772,158.953
C09685=1032.182,346.446,-131.724,172.078,45.771,158.952
C09686=1032.175,346.198,-131.687,172.071,45.769,158.950
C09687=1032.167,345.952,-131.650,172.066,45.768,158.950
C09688=1032.160,345.705,-131.612,172.060,45.767,158.949
C09689=1032.152,345.458,-131.575,172.053,45.765,158.947
C09690=1032.144,345.209,-131.538,172.047,45.764,158.946
C09691=1032.136,344.962,-131.501,172.042,45.762,158.946
C09692=1032.129,344.715,-131.464,172.036,45.760,158.944
C09693=1032.121,344.468,-131.427,172.030,45.759,158.943
C09694=1032.114,344.221,-131.389,172.024,45.758,158.943
C09695=1032.106,343.974,-131.353,172.018,45.756,158.942
C09696=1032.099,343.727,-131.315,172.012,45.755,158.940
C09697=1032.091,343.480,-131.278,172.007,45.753,158.940
C09698=1032.084,343.232,-131.242,172.001,45.752,158.939
C09699=1032.076,342.985,-131.205,171.994,45.751,158.938
C09700=1032.069,342.738,-131.167,171.989,45.749,158.937
C09701=1032.061,342.491,-131.131,171.983,45.747,158.936
C09702=1032.053,342.244,-131.094,171.977,45.746,158.935
C09703=1032.046,341.997,-131.057,171.972,45.745,158.934
C09704=1032.038,341.749,-131.020,171.965,45.744,158.933
C09705=1032.032,341.503,-130.983,171.960,45.742,158.932
C09706=1032.024,341.255,-130.947,171.954,45.741,158.931
C09707=1032.016,341.009,-130.910,171.948,45.740,158.930
C09708=1032.009,340.761,-130.873,171.943,45.738,158.929
C09709=1032.001,340.513,-130.837,171.937,45.737,158.928
C09710=1031.993,340.267,-130.800,171.932,45.736,158.927
C09711=1031.986,340.019,-130.764,171.925,45.734,158.926
C09712=1031.979,339.771,-130.727,171.919,45.733,158.925
C09713=1031.971,339.525,-130.690,171.914,45.732,158.924
C09714=1031.964,339.278,-130.654,171.908,45.730,158.923
C09715=1031.956,339.030,-130.618,171.903,45.730,158.923
C09716=1031.948,338.783,-130.582,171.897,45.728,158.922
C09717=1031.940,338.536,-130.545,171.891,45.727,158.921
C09718=1031.933,338.288,-130.508,171.886,45.726,158.920
C09719=1031.926,338.041,-130.472,171.880,45.725,158.919
C09720=1031.919,337.794,-130.436,171.875,45.724,158.918
C09721=1031.911,337.547,-130.400,171.869,45.722,158.917
C09722=1031.903,337.299,-130.364,171.863,45.721,158.916
C09723=1031.895,337.052,-130.327,171.857,45.720,158.915
C09724=1031.889,336.805,-130.290,171.852,45.719,158.914
C09725=1031.881,336.558,-130.254,171.846,45.718,158.913
C09726=1031.874,336.311,-130.218,171.841,45.716,158.913
C09727=1031.862,335.906,-130.159,171.831,45.715,158.911
C09728=1031.850,335.502,-130.099,171.823,45.713,158.910
C09729=1031.838,335.098,-130.040,171.814,45.711,158.908
C09730=1031.826,334.694,-129.981,171.804,45.709,158.907
C09731=1031.819,334.446,-129.945,171.799,45.708,158.906
C09732=1031.811,334.199,-129.909,171.793,45.707,158.905
C09733=1031.804,333.952,-129.873,171.788,45.706,158.904
C09734=1031.796,333.704,-129.838,171.782,45.705,158.903
C09735=1031.789,333.457,-129.802,171.777,45.704,158.903
C09736=1031.781,333.210,-129.766,171.771,45.703,158.902
C09737=1031.774,332.962,-129.731,171.766,45.702,158.901
C09738=1031.766,332.715,-129.695,171.762,45.701,158.900
C09739=1031.759,332.468,-129.659,171.755,45.700,158.899
C09740=1031.752,332.220,-129.624,171.751,45.699,158.899
C09741=1031.744,331.973,-129.587,171.744,45.698,158.898
C09742=1031.737,331.725,-129.551,171.740,45.697,158.897
C09743=1031.730,331.478,-129.516,171.734,45.696,158.896
C09744=1031.722,331.231,-129.480,171.729,45.695,158.895
C09745=1031.715,330.984,-129.445,171.723,45.694,158.894
C09746=1031.707,330.736,-129.409,171.718,45.693,158.894
C09747=1031.700,330.489,-129.374,171.713,45.692,158.893
C09748=1031.693,330.241,-129.338,171.707,45.691,158.892
C09749=1031.686,329.994,-129.302,171.702,45.690,158.891
C09750=1031.678,329.746,-129.266,171.696,45.690,158.890
C09751=1031.671,329.499,-129.231,171.691,45.688,158.890
C09752=1031.664,329.252,-129.195,171.686,45.687,158.889
C09753=1031.657,329.004,-129.160,171.680,45.687,158.888
C09754=1031.649,328.758,-129.125,171.675,45.686,158.887
C09755=1031.642,328.510,-129.089,171.671,45.685,158.887
C09756=1031.635,328.262,-129.054,171.664,45.684,158.886
C09757=1031.628,328.016,-129.018,171.660,45.683,158.885
C09758=1031.621,327.768,-128.983,171.655,45.682,158.884
C09759=1031.613,327.521,-128.948,171.649,45.681,158.883
C09760=1031.606,327.273,-128.912,171.644,45.680,158.883
C09761=1031.598,327.025,-128.878,171.638,45.680,158.882
C09762=1031.590,326.778,-128.843,171.633,45.679,158.881
C09763=1031.583,326.530,-128.808,171.628,45.678,158.880
C09764=1031.576,326.283,-128.773,171.622,45.677,158.880
C09765=1031.568,326.036,-128.737,171.618,45.677,158.879
C09766=1031.561,325.789,-128.703,171.612,45.676,158.878
C09767=1031.553,325.541,-128.667,171.607,45.676,158.877
C09768=1031.546,325.294,-128.633,171.602,45.675,158.877
C09769=1031.539,325.046,-128.597,171.596,45.674,158.876
C09770=1031.531,324.798,-128.563,171.592,45.673,158.875
C09771=1031.524,324.551,-128.528,171.587,45.672,158.874
C09772=1031.517,324.304,-128.494,171.581,45.672,158.874
C09773=1031.509,324.056,-128.459,171.576,45.671,158.873
C09774=1031.502,323.808,-128.424,171.571,45.671,158.872
C09775=1031.495,323.561,-128.389,171.566,45.670,158.872
C09776=1031.488,323.314,-128.354,171.561,45.669,158.871
C09777=1031.480,323.066,-128.319,171.556,45.668,158.870
C09778=1031.473,322.819,-128.284,171.551,45.668,158.870
C09779=1031.466,322.571,-128.250,171.545,45.667,158.869
C09780=1031.459,322.324,-128.215,171.541,45.666,158.868
C09781=1031.451,322.077,-128.180,171.536,45.665,158.867
C09782=1031.443,321.829,-128.145,171.530,45.665,158.867
C09783=1031.432,321.420,-128.088,171.522,45.664,158.865
C09784=1031.420,321.011,-128.031,171.514,45.663,158.864
C09785=1031.408,320.603,-127.974,171.505,45.662,158.863
C09786=1031.397,320.194,-127.916,171.497,45.661,158.862
C09787=1031.389,319.947,-127.882,171.492,45.660,158.861
C09788=1031.382,319.699,-127.848,171.487,45.660,158.861
C09789=1031.375,319.452,-127.813,171.483,45.659,158.860
C09790=1031.368,319.204,-127.779,171.477,45.659,158.859
C09791=1031.361,318.956,-127.744,171.472,45.658,158.859
C09792=1031.354,318.709,-127.710,171.468,45.658,158.858
C09793=1031.346,318.462,-127.676,171.463,45.657,158.857
C09794=1031.340,318.214,-127.640,171.458,45.656,158.857
C09795=1031.332,317.967,-127.607,171.452,45.656,158.856
C09796=1031.326,317.719,-127.572,171.447,45.655,158.855
C09797=1031.318,317.472,-127.538,171.443,45.655,158.855
C09798=1031.311,317.224,-127.504,171.438,45.654,158.854
C09799=1031.304,316.977,-127.469,171.433,45.654,158.854
C09800=1031.297,316.729,-127.435,171.428,45.653,158.853
C09801=1031.290,316.482,-127.400,171.423,45.653,158.852
C09802=1031.283,316.234,-127.366,171.418,45.652,158.851
C09803=1031.276,315.986,-127.332,171.414,45.652,158.851
C09804=1031.269,315.739,-127.297,171.409,45.651,158.850
C09805=1031.262,315.491,-127.263,171.404,45.651,158.850
C09806=1031.256,315.243,-127.229,171.400,45.650,158.849
C09807=1031.248,314.996,-127.194,171.394,45.650,158.848
C09808=1031.241,314.748,-127.160,171.389,45.649,158.848
C09809=1031.235,314.501,-127.126,171.384,45.649,158.847
C09810=1031.228,314.254,-127.092,171.380,45.648,158.846
C09811=1031.220,314.006,-127.058,171.375,45.648,158.846
C09812=1031.214,313.758,-127.024,171.370,45.647,158.845
C09813=1031.207,313.511,-126.990,171.366,45.647,158.845
C09814=1031.200,313.263,-126.955,171.361,45.647,158.844
C09815=1031.193,313.016,-126.921,171.356,45.646,158.843
C09816=1031.186,312.769,-126.887,171.351,45.646,158.843
C09817=1031.180,312.521,-126.853,171.346,45.645,158.842
C09818=1031.172,312.273,-126.819,171.341,45.645,158.842
C09819=1031.165,312.025,-126.785,171.337,45.644,158.841
C09820=1031.159,311.778,-126.751,171.332,45.644,158.840
C09821=1031.152,311.531,-126.717,171.327,45.644,158.840
C09822=1031.145,311.283,-126.684,171.323,45.643,158.839
C09823=1031.138,311.035,-126.650,171.318,45.642,158.838
C09824=1031.131,310.788,-126.616,171.313,45.642,158.838
C09825=1031.124,310.541,-126.582,171.309,45.642,158.837
C09826=1031.117,310.293,-126.549,171.303,45.642,158.837
C09827=1031.109,310.046,-126.515,171.299,45.642,158.836
C09828=1031.102,309.797,-126.482,171.294,45.641,158.836
C09829=1031.095,309.550,-126.449,171.289,45.641,158.835
C09830=1031.088,309.303,-126.415,171.285,45.641,158.834
C09831=1031.080,309.055,-126.382,171.281,45.641,158.834
C09832=1031.073,308.807,-126.349,171.276,45.641,158.833
C09833=1031.066,308.559,-126.315,171.271,45.641,158.833
C09834=1031.060,308.312,-126.281,171.267,45.640,158.832
C09835=1031.052,308.064,-126.249,171.261,45.640,158.832
C09836=1031.045,307.817,-126.215,171.257,45.640,158.831
C09837=1031.038,307.570,-126.182,171.252,45.640,158.831
C09838=1031.031,307.321,-126.148,171.247,45.639,158.830
C09839=1031.020,306.918,-126.094,171.241,45.639,158.829
C09840=1031.007,306.513,-126.040,171.233,45.639,158.828
C09841=1030.996,306.110,-125.986,171.225,45.639,158.827
C09842=1030.985,305.706,-125.931,171.218,45.638,158.827
C09843=1030.977,305.458,-125.899,171.213,45.638,158.826
C09844=1030.971,305.211,-125.865,171.209,45.638,158.826
C09845=1030.964,304.963,-125.832,171.204,45.638,158.825
C09846=1030.957,304.716,-125.799,171.200,45.638,158.824
C09847=1030.950,304.468,-125.766,171.195,45.637,158.824
C09848=1030.943,304.220,-125.733,171.191,45.638,158.824
C09849=1030.936,303.973,-125.700,171.186,45.637,158.823
C09850=1030.929,303.725,-125.667,171.182,45.637,158.822
C09851=1030.922,303.478,-125.634,171.176,45.637,158.822
C09852=1030.915,303.229,-125.601,171.172,45.637,158.821
C09853=1030.909,302.982,-125.568,171.168,45.637,158.821
C09854=1030.901,302.734,-125.535,171.164,45.637,158.820
C09855=1030.894,302.487,-125.502,171.159,45.637,158.820
C09856=1030.888,302.238,-125.469,171.155,45.637,158.819
C09857=1030.881,301.992,-125.435,171.150,45.636,158.819
C09858=1030.873,301.744,-125.403,171.146,45.636,158.818
C09859=1030.867,301.496,-125.370,171.141,45.636,158.818
C09860=1030.860,301.248,-125.337,171.137,45.636,158.817
C09861=1030.853,301.001,-125.304,171.133,45.637,158.817
C09862=1030.846,300.753,-125.271,171.128,45.636,158.816
C09863=1030.840,300.505,-125.238,171.123,45.636,158.816
C09864=1030.832,300.257,-125.206,171.119,45.636,158.815
C09865=1030.826,300.010,-125.173,171.114,45.636,158.815
C09866=1030.819,299.761,-125.140,171.110,45.636,158.814
C09867=1030.812,299.514,-125.106,171.106,45.636,158.814
C09868=1030.805,299.267,-125.074,171.101,45.636,158.813
C09869=1030.798,299.019,-125.041,171.097,45.636,158.813
C09870=1030.792,298.771,-125.008,171.092,45.636,158.812
C09871=1030.784,298.523,-124.976,171.088,45.636,158.812
C09872=1030.778,298.276,-124.943,171.083,45.636,158.811
C09873=1030.772,298.028,-124.910,171.080,45.636,158.811
C09874=1030.764,297.780,-124.878,171.075,45.636,158.811
C09875=1030.758,297.532,-124.845,171.071,45.636,158.810
C09876=1030.752,297.285,-124.812,171.066,45.636,158.810
C09877=1030.745,297.036,-124.779,171.062,45.636,158.809
C09878=1030.738,296.789,-124.747,171.058,45.636,158.809
C09879=1030.731,296.542,-124.714,171.053,45.636,158.808
C09880=1030.724,296.293,-124.681,171.049,45.636,158.808
C09881=1030.717,296.046,-124.649,171.044,45.636,158.807
C09882=1030.711,295.798,-124.616,171.041,45.636,158.807
C09883=1030.705,295.551,-124.584,171.036,45.636,158.806
C09884=1030.697,295.303,-124.551,171.032,45.636,158.806
C09885=1030.691,295.055,-124.518,171.028,45.636,158.805
C09886=1030.685,294.807,-124.486,171.023,45.636,158.805
C09887=1030.678,294.560,-124.454,171.019,45.636,158.804
C09888=1030.671,294.311,-124.421,171.014,45.636,158.804
C09889=1030.664,294.064,-124.389,171.011,45.636,158.804
C09890=1030.658,293.816,-124.357,171.006,45.636,158.803
C09891=1030.650,293.568,-124.324,171.002,45.637,158.803
C09892=1030.643,293.321,-124.292,170.998,45.637,158.802
C09893=1030.637,293.072,-124.260,170.993,45.637,158.802
C09894=1030.630,292.825,-124.228,170.989,45.637,158.801
C09895=1030.620,292.438,-124.178,170.982,45.637,158.801
C09896=1030.608,292.051,-124.128,170.976,45.637,158.800
C09897=1030.598,291.664,-124.078,170.969,45.638,158.800
C09898=1030.587,291.278,-124.027,170.963,45.638,158.799
C09899=1030.580,291.030,-123.996,170.958,45.639,158.799
C09900=1030.574,290.782,-123.964,170.954,45.639,158.798
C09901=1030.567,290.534,-123.932,170.950,45.639,158.798
C09902=1030.560,290.286,-123.900,170.946,45.639,158.797
C09903=1030.553,290.038,-123.868,170.942,45.639,158.797
C09904=1030.546,289.791,-123.836,170.938,45.639,158.796
C09905=1030.540,289.543,-123.804,170.933,45.640,158.796
C09906=1030.533,289.295,-123.772,170.929,45.640,158.796
C09907=1030.526,289.047,-123.741,170.925,45.640,158.795
C09908=1030.519,288.800,-123.709,170.921,45.640,158.795
C09909=1030.512,288.551,-123.677,170.917,45.641,158.795
C09910=1030.506,288.303,-123.645,170.913,45.641,158.794
C09911=1030.499,288.056,-123.613,170.909,45.641,158.794
C09912=1030.492,287.808,-123.581,170.904,45.642,158.793
C09913=1030.486,287.560,-123.550,170.901,45.642,158.793
C09914=1030.479,287.312,-123.518,170.897,45.642,158.793
C09915=1030.472,287.065,-123.486,170.892,45.643,158.792
C09916=1030.465,286.817,-123.455,170.888,45.643,158.792
C09917=1030.458,286.569,-123.423,170.884,45.643,158.791
C09918=1030.452,286.321,-123.391,170.880,45.643,158.791
C09919=1030.445,286.073,-123.359,170.876,45.644,158.791
C09920=1030.438,285.825,-123.327,170.872,45.644,158.790
C09921=1030.431,285.577,-123.296,170.867,45.644,158.790
C09922=1030.424,285.329,-123.265,170.863,45.645,158.790
C09923=1030.417,285.081,-123.234,170.859,45.646,158.789
C09924=1030.410,284.834,-123.202,170.856,45.646,158.789
C09925=1030.404,284.586,-123.171,170.851,45.646,158.789
C09926=1030.397,284.338,-123.139,170.847,45.646,158.788
C09927=1030.390,284.090,-123.108,170.843,45.647,158.788
C09928=1030.383,283.842,-123.076,170.840,45.647,158.788
C09929=1030.377,283.594,-123.045,170.835,45.648,158.787
C09930=1030.370,283.346,-123.014,170.831,45.648,158.787
C09931=1030.363,283.098,-122.982,170.827,45.648,158.786
C09932=1030.357,282.850,-122.951,170.823,45.649,158.786
C09933=1030.350,282.602,-122.919,170.819,45.649,158.786
C09934=1030.342,282.355,-122.888,170.815,45.650,158.786
C09935=1030.336,282.106,-122.858,170.811,45.650,158.785
C09936=1030.329,281.858,-122.826,170.807,45.650,158.785
C09937=1030.323,281.611,-122.795,170.804,45.651,158.785
C09938=1030.316,281.363,-122.763,170.799,45.651,158.784
C09939=1030.309,281.115,-122.732,170.795,45.652,158.784
C09940=1030.302,280.867,-122.701,170.791,45.653,158.784
C09941=1030.296,280.619,-122.669,170.788,45.653,158.783
C09942=1030.289,280.370,-122.638,170.783,45.653,158.783
C09943=1030.282,280.122,-122.607,170.779,45.654,158.782
C09944=1030.275,279.875,-122.576,170.775,45.654,158.782
C09945=1030.268,279.627,-122.545,170.772,45.655,158.782
C09946=1030.262,279.380,-122.514,170.767,45.655,158.781
C09947=1030.256,279.131,-122.483,170.763,45.656,158.781
C09948=1030.249,278.883,-122.451,170.760,45.656,158.781
C09949=1030.242,278.635,-122.420,170.756,45.656,158.781
C09950=1030.236,278.387,-122.389,170.752,45.657,158.780
C09951=1030.226,278.012,-122.342,170.746,45.658,158.780
C09952=1030.215,277.638,-122.296,170.740,45.659,158.779
C09953=1030.205,277.263,-122.248,170.734,45.659,158.779
C09954=1030.195,276.888,-122.202,170.728,45.660,158.778
C09955=1030.189,276.641,-122.171,170.724,45.661,158.778
C09956=1030.182,276.392,-122.141,170.720,45.661,158.778
C09957=1030.175,276.145,-122.110,170.717,45.662,158.778
C09958=1030.168,275.896,-122.079,170.713,45.662,158.777
C09959=1030.162,275.648,-122.048,170.709,45.663,158.777
C09960=1030.154,275.400,-122.017,170.705,45.663,158.777
C09961=1030.148,275.153,-121.986,170.701,45.664,158.776
C09962=1030.142,274.905,-121.956,170.697,45.665,158.776
C09963=1030.134,274.657,-121.925,170.693,45.666,158.776
C09964=1030.128,274.408,-121.894,170.690,45.666,158.775
C09965=1030.121,274.160,-121.864,170.685,45.667,158.775
C09966=1030.115,273.913,-121.833,170.681,45.668,158.775
C09967=1030.108,273.664,-121.802,170.678,45.668,158.775
C09968=1030.101,273.417,-121.771,170.674,45.669,158.774
C09969=1030.094,273.168,-121.741,170.670,45.669,158.774
C09970=1030.088,272.921,-121.711,170.667,45.670,158.774
C09971=1030.081,272.672,-121.680,170.663,45.671,158.774
C09972=1030.075,272.424,-121.649,170.658,45.671,158.773
C09973=1030.068,272.176,-121.619,170.655,45.672,158.773
C09974=1030.062,271.928,-121.588,170.651,45.673,158.773
C09975=1030.054,271.681,-121.557,170.647,45.673,158.772
C09976=1030.048,271.432,-121.527,170.644,45.674,158.772
C09977=1030.041,271.184,-121.497,170.640,45.674,158.772
C09978=1030.035,270.936,-121.466,170.637,45.675,158.772
C09979=1030.028,270.688,-121.436,170.633,45.676,158.771
C09980=1030.021,270.440,-121.405,170.629,45.677,158.771
C09981=1030.014,270.193,-121.375,170.625,45.677,158.771
C09982=1030.008,269.944,-121.344,170.621,45.678,158.771
C09983=1030.001,269.696,-121.314,170.617,45.679,158.770
C09984=1029.994,269.448,-121.284,170.614,45.679,158.770
C09985=1029.988,269.200,-121.254,170.610,45.680,158.770
C09986=1029.981,268.952,-121.224,170.606,45.681,158.770
C09987=1029.974,268.703,-121.193,170.603,45.681,158.770
C09988=1029.968,268.456,-121.163,170.599,45.682,158.769
C09989=1029.961,268.207,-121.133,170.594,45.683,158.769
C09990=1029.955,267.960,-121.103,170.591,45.683,158.769
C09991=1029.948,267.711,-121.072,170.587,45.684,158.768
C09992=1029.941,267.463,-121.042,170.584,45.685,158.768
C09993=1029.935,267.215,-121.012,170.580,45.686,158.768
C09994=1029.927,266.967,-120.982,170.576,45.687,158.768
C09995=1029.921,266.719,-120.951,170.573,45.687,158.768
C09996=1029.914,266.471,-120.921,170.569,45.688,158.767
//INST
///DATE 2021/06/17 10:58
///ATTR SC,RW,RJ
////FRAME ROBOT
///GROUP1 RB1
NOP
MOVL C00000 V=800.0 PL=0
MOVL C00001 V=800.0 PL=0
MOVL C00002 V=800.0 PL=0
MOVL C00003 V=800.0 PL=0
MOVL C00004 V=800.0 PL=0
MOVL C00005 V=800.0 PL=0
MOVL C00006 V=800.0 PL=0
MOVL C00007 V=800.0 PL=0
MOVL C00008 V=800.0 PL=0
MOVL C00009 V=800.0 PL=0
MOVL C00010 V=800.0 PL=0
MOVL C00011 V=800.0 PL=0
MOVL C00012 V=800.0 PL=0
MOVL C00013 V=800.0 PL=0
MOVL C00014 V=800.0 PL=0
MOVL C00015 V=800.0 PL=0
MOVL C00016 V=800.0 PL=0
MOVL C00017 V=800.0 PL=0
MOVL C00018 V=800.0 PL=0
MOVL C00019 V=800.0 PL=0
MOVL C00020 V=800.0 PL=0
MOVL C00021 V=800.0 PL=0
MOVL C00022 V=800.0 PL=0
MOVL C00023 V=800.0 PL=0
MOVL C00024 V=800.0 PL=0
MOVL C00025 V=800.0 PL=0
MOVL C00026 V=800.0 PL=0
MOVL C00027 V=800.0 PL=0
MOVL C00028 V=800.0 PL=0
MOVL C00029 V=800.0 PL=0
MOVL C00030 V=800.0 PL=0
MOVL C00031 V=800.0 PL=0
MOVL C00032 V=800.0 PL=0
MOVL C00033 V=800.0 PL=0
MOVL C00034 V=800.0 PL=0
MOVL C00035 V=800.0 PL=0
MOVL C00036 V=800.0 PL=0
MOVL C00037 V=800.0 PL=0
MOVL C00038 V=800.0 PL=0
MOVL C00039 V=800.0 PL=0
MOVL C00040 V=800.0 PL=0
MOVL C00041 V=800.0 PL=0
MOVL C00042 V=800.0 PL=0
MOVL C00043 V=800.0 PL=0
MOVL C00044 V=800.0 PL=0
MOVL C00045 V=800.0 PL=0
MOVL C00046 V=800.0 PL=0
MOVL C00047 V=800.0 PL=0
MOVL C00048 V=800.0 PL=0
MOVL C00049 V=800.0 PL=0
MOVL C00050 V=800.0 PL=0
MOVL C00051 V=800.0 PL=0
MOVL C00052 V=800.0 PL=0
MOVL C00053 V=800.0 PL=0
MOVL C00054 V=800.0 PL=0
MOVL C00055 V=800.0 PL=0
MOVL C00056 V=800.0 PL=0
MOVL C00057 V=800.0 PL=0
MOVL C00058 V=800.0 PL=0
MOVL C00059 V=800.0 PL=0
MOVL C00060 V=800.0 PL=0
MOVL C00061 V=800.0 PL=0
MOVL C00062 V=800.0 PL=0
MOVL C00063 V=800.0 PL=0
MOVL C00064 V=800.0 PL=0
MOVL C00065 V=800.0 PL=0
MOVL C00066 V=800.0 PL=0
MOVL C00067 V=800.0 PL=0
MOVL C00068 V=800.0 PL=0
MOVL C00069 V=800.0 PL=0
MOVL C00070 V=800.0 PL=0
MOVL C00071 V=800.0 PL=0
MOVL C00072 V=800.0 PL=0
MOVL C00073 V=800.0 PL=0
MOVL C00074 V=800.0 PL=0
MOVL C00075 V=800.0 PL=0
MOVL C00076 V=800.0 PL=0
MOVL C00077 V=800.0 PL=0
MOVL C00078 V=800.0 PL=0
MOVL C00079 V=800.0 PL=0
MOVL C00080 V=800.0 PL=0
MOVL C00081 V=800.0 PL=0
MOVL C00082 V=800.0 PL=0
MOVL C00083 V=800.0 PL=0
MOVL C00084 V=800.0 PL=0
MOVL C00085 V=800.0 PL=0
MOVL C00086 V=800.0 PL=0
MOVL C00087 V=800.0 PL=0
MOVL C00088 V=800.0 PL=0
MOVL C00089 V=800.0 PL=0
MOVL C00090 V=800.0 PL=0
MOVL C00091 V=800.0 PL=0
MOVL C00092 V=800.0 PL=0
MOVL C00093 V=800.0 PL=0
MOVL C00094 V=800.0 PL=0
MOVL C00095 V=800.0 PL=0
MOVL C00096 V=800.0 PL=0
MOVL C00097 V=800.0 PL=0
MOVL C00098 V=800.0 PL=0
MOVL C00099 V=800.0 PL=0
MOVL C00100 V=800.0 PL=0
MOVL C00101 V=800.0 PL=0
MOVL C00102 V=800.0 PL=0
MOVL C00103 V=800.0 PL=0
MOVL C00104 V=800.0 PL=0
MOVL C00105 V=800.0 PL=0
MOVL C00106 V=800.0 PL=0
MOVL C00107 V=800.0 PL=0
MOVL C00108 V=800.0 PL=0
MOVL C00109 V=800.0 PL=0
MOVL C00110 V=800.0 PL=0
MOVL C00111 V=800.0 PL=0
MOVL C00112 V=800.0 PL=0
MOVL C00113 V=800.0 PL=0
MOVL C00114 V=800.0 PL=0
MOVL C00115 V=800.0 PL=0
MOVL C00116 V=800.0 PL=0
MOVL C00117 V=800.0 PL=0
MOVL C00118 V=800.0 PL=0
MOVL C00119 V=800.0 PL=0
MOVL C00120 V=800.0 PL=0
MOVL C00121 V=800.0 PL=0
MOVL C00122 V=800.0 PL=0
MOVL C00123 V=800.0 PL=0
MOVL C00124 V=800.0 PL=0
MOVL C00125 V=800.0 PL=0
MOVL C00126 V=800.0 PL=0
MOVL C00127 V=800.0 PL=0
MOVL C00128 V=800.0 PL=0
MOVL C00129 V=800.0 PL=0
MOVL C00130 V=800.0 PL=0
MOVL C00131 V=800.0 PL=0
MOVL C00132 V=800.0 PL=0
MOVL C00133 V=800.0 PL=0
MOVL C00134 V=800.0 PL=0
MOVL C00135 V=800.0 PL=0
MOVL C00136 V=800.0 PL=0
MOVL C00137 V=800.0 PL=0
MOVL C00138 V=800.0 PL=0
MOVL C00139 V=800.0 PL=0
MOVL C00140 V=800.0 PL=0
MOVL C00141 V=800.0 PL=0
MOVL C00142 V=800.0 PL=0
MOVL C00143 V=800.0 PL=0
MOVL C00144 V=800.0 PL=0
MOVL C00145 V=800.0 PL=0
MOVL C00146 V=800.0 PL=0
MOVL C00147 V=800.0 PL=0
MOVL C00148 V=800.0 PL=0
MOVL C00149 V=800.0 PL=0
MOVL C00150 V=800.0 PL=0
MOVL C00151 V=800.0 PL=0
MOVL C00152 V=800.0 PL=0
MOVL C00153 V=800.0 PL=0
MOVL C00154 V=800.0 PL=0
MOVL C00155 V=800.0 PL=0
MOVL C00156 V=800.0 PL=0
MOVL C00157 V=800.0 PL=0
MOVL C00158 V=800.0 PL=0
MOVL C00159 V=800.0 PL=0
MOVL C00160 V=800.0 PL=0
MOVL C00161 V=800.0 PL=0
MOVL C00162 V=800.0 PL=0
MOVL C00163 V=800.0 PL=0
MOVL C00164 V=800.0 PL=0
MOVL C00165 V=800.0 PL=0
MOVL C00166 V=800.0 PL=0
MOVL C00167 V=800.0 PL=0
MOVL C00168 V=800.0 PL=0
MOVL C00169 V=800.0 PL=0
MOVL C00170 V=800.0 PL=0
MOVL C00171 V=800.0 PL=0
MOVL C00172 V=800.0 PL=0
MOVL C00173 V=800.0 PL=0
MOVL C00174 V=800.0 PL=0
MOVL C00175 V=800.0 PL=0
MOVL C00176 V=800.0 PL=0
MOVL C00177 V=800.0 PL=0
MOVL C00178 V=800.0 PL=0
MOVL C00179 V=800.0 PL=0
MOVL C00180 V=800.0 PL=0
MOVL C00181 V=800.0 PL=0
MOVL C00182 V=800.0 PL=0
MOVL C00183 V=800.0 PL=0
MOVL C00184 V=800.0 PL=0
MOVL C00185 V=800.0 PL=0
MOVL C00186 V=800.0 PL=0
MOVL C00187 V=800.0 PL=0
MOVL C00188 V=800.0 PL=0
MOVL C00189 V=800.0 PL=0
MOVL C00190 V=800.0 PL=0
MOVL C00191 V=800.0 PL=0
MOVL C00192 V=800.0 PL=0
MOVL C00193 V=800.0 PL=0
MOVL C00194 V=800.0 PL=0
MOVL C00195 V=800.0 PL=0
MOVL C00196 V=800.0 PL=0
MOVL C00197 V=800.0 PL=0
MOVL C00198 V=800.0 PL=0
MOVL C00199 V=800.0 PL=0
MOVL C00200 V=800.0 PL=0
MOVL C00201 V=800.0 PL=0
MOVL C00202 V=800.0 PL=0
MOVL C00203 V=800.0 PL=0
MOVL C00204 V=800.0 PL=0
MOVL C00205 V=800.0 PL=0
MOVL C00206 V=800.0 PL=0
MOVL C00207 V=800.0 PL=0
MOVL C00208 V=800.0 PL=0
MOVL C00209 V=800.0 PL=0
MOVL C00210 V=800.0 PL=0
MOVL C00211 V=800.0 PL=0
MOVL C00212 V=800.0 PL=0
MOVL C00213 V=800.0 PL=0
MOVL C00214 V=800.0 PL=0
MOVL C00215 V=800.0 PL=0
MOVL C00216 V=800.0 PL=0
MOVL C00217 V=800.0 PL=0
MOVL C00218 V=800.0 PL=0
MOVL C00219 V=800.0 PL=0
MOVL C00220 V=800.0 PL=0
MOVL C00221 V=800.0 PL=0
MOVL C00222 V=800.0 PL=0
MOVL C00223 V=800.0 PL=0
MOVL C00224 V=800.0 PL=0
MOVL C00225 V=800.0 PL=0
MOVL C00226 V=800.0 PL=0
MOVL C00227 V=800.0 PL=0
MOVL C00228 V=800.0 PL=0
MOVL C00229 V=800.0 PL=0
MOVL C00230 V=800.0 PL=0
MOVL C00231 V=800.0 PL=0
MOVL C00232 V=800.0 PL=0
MOVL C00233 V=800.0 PL=0
MOVL C00234 V=800.0 PL=0
MOVL C00235 V=800.0 PL=0
MOVL C00236 V=800.0 PL=0
MOVL C00237 V=800.0 PL=0
MOVL C00238 V=800.0 PL=0
MOVL C00239 V=800.0 PL=0
MOVL C00240 V=800.0 PL=0
MOVL C00241 V=800.0 PL=0
MOVL C00242 V=800.0 PL=0
MOVL C00243 V=800.0 PL=0
MOVL C00244 V=800.0 PL=0
MOVL C00245 V=800.0 PL=0
MOVL C00246 V=800.0 PL=0
MOVL C00247 V=800.0 PL=0
MOVL C00248 V=800.0 PL=0
MOVL C00249 V=800.0 PL=0
MOVL C00250 V=800.0 PL=0
MOVL C00251 V=800.0 PL=0
MOVL C00252 V=800.0 PL=0
MOVL C00253 V=800.0 PL=0
MOVL C00254 V=800.0 PL=0
MOVL C00255 V=800.0 PL=0
MOVL C00256 V=800.0 PL=0
MOVL C00257 V=800.0 PL=0
MOVL C00258 V=800.0 PL=0
MOVL C00259 V=800.0 PL=0
MOVL C00260 V=800.0 PL=0
MOVL C00261 V=800.0 PL=0
MOVL C00262 V=800.0 PL=0
MOVL C00263 V=800.0 PL=0
MOVL C00264 V=800.0 PL=0
MOVL C00265 V=800.0 PL=0
MOVL C00266 V=800.0 PL=0
MOVL C00267 V=800.0 PL=0
MOVL C00268 V=800.0 PL=0
MOVL C00269 V=800.0 PL=0
MOVL C00270 V=800.0 PL=0
MOVL C00271 V=800.0 PL=0
MOVL C00272 V=800.0 PL=0
MOVL C00273 V=800.0 PL=0
MOVL C00274 V=800.0 PL=0
MOVL C00275 V=800.0 PL=0
MOVL C00276 V=800.0 PL=0
MOVL C00277 V=800.0 PL=0
MOVL C00278 V=800.0 PL=0
MOVL C00279 V=800.0 PL=0
MOVL C00280 V=800.0 PL=0
MOVL C00281 V=800.0 PL=0
MOVL C00282 V=800.0 PL=0
MOVL C00283 V=800.0 PL=0
MOVL C00284 V=800.0 PL=0
MOVL C00285 V=800.0 PL=0
MOVL C00286 V=800.0 PL=0
MOVL C00287 V=800.0 PL=0
MOVL C00288 V=800.0 PL=0
MOVL C00289 V=800.0 PL=0
MOVL C00290 V=800.0 PL=0
MOVL C00291 V=800.0 PL=0
MOVL C00292 V=800.0 PL=0
MOVL C00293 V=800.0 PL=0
MOVL C00294 V=800.0 PL=0
MOVL C00295 V=800.0 PL=0
MOVL C00296 V=800.0 PL=0
MOVL C00297 V=800.0 PL=0
MOVL C00298 V=800.0 PL=0
MOVL C00299 V=800.0 PL=0
MOVL C00300 V=800.0 PL=0
MOVL C00301 V=800.0 PL=0
MOVL C00302 V=800.0 PL=0
MOVL C00303 V=800.0 PL=0
MOVL C00304 V=800.0 PL=0
MOVL C00305 V=800.0 PL=0
MOVL C00306 V=800.0 PL=0
MOVL C00307 V=800.0 PL=0
MOVL C00308 V=800.0 PL=0
MOVL C00309 V=800.0 PL=0
MOVL C00310 V=800.0 PL=0
MOVL C00311 V=800.0 PL=0
MOVL C00312 V=800.0 PL=0
MOVL C00313 V=800.0 PL=0
MOVL C00314 V=800.0 PL=0
MOVL C00315 V=800.0 PL=0
MOVL C00316 V=800.0 PL=0
MOVL C00317 V=800.0 PL=0
MOVL C00318 V=800.0 PL=0
MOVL C00319 V=800.0 PL=0
MOVL C00320 V=800.0 PL=0
MOVL C00321 V=800.0 PL=0
MOVL C00322 V=800.0 PL=0
MOVL C00323 V=800.0 PL=0
MOVL C00324 V=800.0 PL=0
MOVL C00325 V=800.0 PL=0
MOVL C00326 V=800.0 PL=0
MOVL C00327 V=800.0 PL=0
MOVL C00328 V=800.0 PL=0
MOVL C00329 V=800.0 PL=0
MOVL C00330 V=800.0 PL=0
MOVL C00331 V=800.0 PL=0
MOVL C00332 V=800.0 PL=0
MOVL C00333 V=800.0 PL=0
MOVL C00334 V=800.0 PL=0
MOVL C00335 V=800.0 PL=0
MOVL C00336 V=800.0 PL=0
MOVL C00337 V=800.0 PL=0
MOVL C00338 V=800.0 PL=0
MOVL C00339 V=800.0 PL=0
MOVL C00340 V=800.0 PL=0
MOVL C00341 V=800.0 PL=0
MOVL C00342 V=800.0 PL=0
MOVL C00343 V=800.0 PL=0
MOVL C00344 V=800.0 PL=0
MOVL C00345 V=800.0 PL=0
MOVL C00346 V=800.0 PL=0
MOVL C00347 V=800.0 PL=0
MOVL C00348 V=800.0 PL=0
MOVL C00349 V=800.0 PL=0
MOVL C00350 V=800.0 PL=0
MOVL C00351 V=800.0 PL=0
MOVL C00352 V=800.0 PL=0
MOVL C00353 V=800.0 PL=0
MOVL C00354 V=800.0 PL=0
MOVL C00355 V=800.0 PL=0
MOVL C00356 V=800.0 PL=0
MOVL C00357 V=800.0 PL=0
MOVL C00358 V=800.0 PL=0
MOVL C00359 V=800.0 PL=0
MOVL C00360 V=800.0 PL=0
MOVL C00361 V=800.0 PL=0
MOVL C00362 V=800.0 PL=0
MOVL C00363 V=800.0 PL=0
MOVL C00364 V=800.0 PL=0
MOVL C00365 V=800.0 PL=0
MOVL C00366 V=800.0 PL=0
MOVL C00367 V=800.0 PL=0
MOVL C00368 V=800.0 PL=0
MOVL C00369 V=800.0 PL=0
MOVL C00370 V=800.0 PL=0
MOVL C00371 V=800.0 PL=0
MOVL C00372 V=800.0 PL=0
MOVL C00373 V=800.0 PL=0
MOVL C00374 V=800.0 PL=0
MOVL C00375 V=800.0 PL=0
MOVL C00376 V=800.0 PL=0
MOVL C00377 V=800.0 PL=0
MOVL C00378 V=800.0 PL=0
MOVL C00379 V=800.0 PL=0
MOVL C00380 V=800.0 PL=0
MOVL C00381 V=800.0 PL=0
MOVL C00382 V=800.0 PL=0
MOVL C00383 V=800.0 PL=0
MOVL C00384 V=800.0 PL=0
MOVL C00385 V=800.0 PL=0
MOVL C00386 V=800.0 PL=0
MOVL C00387 V=800.0 PL=0
MOVL C00388 V=800.0 PL=0
MOVL C00389 V=800.0 PL=0
MOVL C00390 V=800.0 PL=0
MOVL C00391 V=800.0 PL=0
MOVL C00392 V=800.0 PL=0
MOVL C00393 V=800.0 PL=0
MOVL C00394 V=800.0 PL=0
MOVL C00395 V=800.0 PL=0
MOVL C00396 V=800.0 PL=0
MOVL C00397 V=800.0 PL=0
MOVL C00398 V=800.0 PL=0
MOVL C00399 V=800.0 PL=0
MOVL C00400 V=800.0 PL=0
MOVL C00401 V=800.0 PL=0
MOVL C00402 V=800.0 PL=0
MOVL C00403 V=800.0 PL=0
MOVL C00404 V=800.0 PL=0
MOVL C00405 V=800.0 PL=0
MOVL C00406 V=800.0 PL=0
MOVL C00407 V=800.0 PL=0
MOVL C00408 V=800.0 PL=0
MOVL C00409 V=800.0 PL=0
MOVL C00410 V=800.0 PL=0
MOVL C00411 V=800.0 PL=0
MOVL C00412 V=800.0 PL=0
MOVL C00413 V=800.0 PL=0
MOVL C00414 V=800.0 PL=0
MOVL C00415 V=800.0 PL=0
MOVL C00416 V=800.0 PL=0
MOVL C00417 V=800.0 PL=0
MOVL C00418 V=800.0 PL=0
MOVL C00419 V=800.0 PL=0
MOVL C00420 V=800.0 PL=0
MOVL C00421 V=800.0 PL=0
MOVL C00422 V=800.0 PL=0
MOVL C00423 V=800.0 PL=0
MOVL C00424 V=800.0 PL=0
MOVL C00425 V=800.0 PL=0
MOVL C00426 V=800.0 PL=0
MOVL C00427 V=800.0 PL=0
MOVL C00428 V=800.0 PL=0
MOVL C00429 V=800.0 PL=0
MOVL C00430 V=800.0 PL=0
MOVL C00431 V=800.0 PL=0
MOVL C00432 V=800.0 PL=0
MOVL C00433 V=800.0 PL=0
MOVL C00434 V=800.0 PL=0
MOVL C00435 V=800.0 PL=0
MOVL C00436 V=800.0 PL=0
MOVL C00437 V=800.0 PL=0
MOVL C00438 V=800.0 PL=0
MOVL C00439 V=800.0 PL=0
MOVL C00440 V=800.0 PL=0
MOVL C00441 V=800.0 PL=0
MOVL C00442 V=800.0 PL=0
MOVL C00443 V=800.0 PL=0
MOVL C00444 V=800.0 PL=0
MOVL C00445 V=800.0 PL=0
MOVL C00446 V=800.0 PL=0
MOVL C00447 V=800.0 PL=0
MOVL C00448 V=800.0 PL=0
MOVL C00449 V=800.0 PL=0
MOVL C00450 V=800.0 PL=0
MOVL C00451 V=800.0 PL=0
MOVL C00452 V=800.0 PL=0
MOVL C00453 V=800.0 PL=0
MOVL C00454 V=800.0 PL=0
MOVL C00455 V=800.0 PL=0
MOVL C00456 V=800.0 PL=0
MOVL C00457 V=800.0 PL=0
MOVL C00458 V=800.0 PL=0
MOVL C00459 V=800.0 PL=0
MOVL C00460 V=800.0 PL=0
MOVL C00461 V=800.0 PL=0
MOVL C00462 V=800.0 PL=0
MOVL C00463 V=800.0 PL=0
MOVL C00464 V=800.0 PL=0
MOVL C00465 V=800.0 PL=0
MOVL C00466 V=800.0 PL=0
MOVL C00467 V=800.0 PL=0
MOVL C00468 V=800.0 PL=0
MOVL C00469 V=800.0 PL=0
MOVL C00470 V=800.0 PL=0
MOVL C00471 V=800.0 PL=0
MOVL C00472 V=800.0 PL=0
MOVL C00473 V=800.0 PL=0
MOVL C00474 V=800.0 PL=0
MOVL C00475 V=800.0 PL=0
MOVL C00476 V=800.0 PL=0
MOVL C00477 V=800.0 PL=0
MOVL C00478 V=800.0 PL=0
MOVL C00479 V=800.0 PL=0
MOVL C00480 V=800.0 PL=0
MOVL C00481 V=800.0 PL=0
MOVL C00482 V=800.0 PL=0
MOVL C00483 V=800.0 PL=0
MOVL C00484 V=800.0 PL=0
MOVL C00485 V=800.0 PL=0
MOVL C00486 V=800.0 PL=0
MOVL C00487 V=800.0 PL=0
MOVL C00488 V=800.0 PL=0
MOVL C00489 V=800.0 PL=0
MOVL C00490 V=800.0 PL=0
MOVL C00491 V=800.0 PL=0
MOVL C00492 V=800.0 PL=0
MOVL C00493 V=800.0 PL=0
MOVL C00494 V=800.0 PL=0
MOVL C00495 V=800.0 PL=0
MOVL C00496 V=800.0 PL=0
MOVL C00497 V=800.0 PL=0
MOVL C00498 V=800.0 PL=0
MOVL C00499 V=800.0 PL=0
MOVL C00500 V=800.0 PL=0
MOVL C00501 V=800.0 PL=0
MOVL C00502 V=800.0 PL=0
MOVL C00503 V=800.0 PL=0
MOVL C00504 V=800.0 PL=0
MOVL C00505 V=800.0 PL=0
MOVL C00506 V=800.0 PL=0
MOVL C00507 V=800.0 PL=0
MOVL C00508 V=800.0 PL=0
MOVL C00509 V=800.0 PL=0
MOVL C00510 V=800.0 PL=0
MOVL C00511 V=800.0 PL=0
MOVL C00512 V=800.0 PL=0
MOVL C00513 V=800.0 PL=0
MOVL C00514 V=800.0 PL=0
MOVL C00515 V=800.0 PL=0
MOVL C00516 V=800.0 PL=0
MOVL C00517 V=800.0 PL=0
MOVL C00518 V=800.0 PL=0
MOVL C00519 V=800.0 PL=0
MOVL C00520 V=800.0 PL=0
MOVL C00521 V=800.0 PL=0
MOVL C00522 V=800.0 PL=0
MOVL C00523 V=800.0 PL=0
MOVL C00524 V=800.0 PL=0
MOVL C00525 V=800.0 PL=0
MOVL C00526 V=800.0 PL=0
MOVL C00527 V=800.0 PL=0
MOVL C00528 V=800.0 PL=0
MOVL C00529 V=800.0 PL=0
MOVL C00530 V=800.0 PL=0
MOVL C00531 V=800.0 PL=0
MOVL C00532 V=800.0 PL=0
MOVL C00533 V=800.0 PL=0
MOVL C00534 V=800.0 PL=0
MOVL C00535 V=800.0 PL=0
MOVL C00536 V=800.0 PL=0
MOVL C00537 V=800.0 PL=0
MOVL C00538 V=800.0 PL=0
MOVL C00539 V=800.0 PL=0
MOVL C00540 V=800.0 PL=0
MOVL C00541 V=800.0 PL=0
MOVL C00542 V=800.0 PL=0
MOVL C00543 V=800.0 PL=0
MOVL C00544 V=800.0 PL=0
MOVL C00545 V=800.0 PL=0
MOVL C00546 V=800.0 PL=0
MOVL C00547 V=800.0 PL=0
MOVL C00548 V=800.0 PL=0
MOVL C00549 V=800.0 PL=0
MOVL C00550 V=800.0 PL=0
MOVL C00551 V=800.0 PL=0
MOVL C00552 V=800.0 PL=0
MOVL C00553 V=800.0 PL=0
MOVL C00554 V=800.0 PL=0
MOVL C00555 V=800.0 PL=0
MOVL C00556 V=800.0 PL=0
MOVL C00557 V=800.0 PL=0
MOVL C00558 V=800.0 PL=0
MOVL C00559 V=800.0 PL=0
MOVL C00560 V=800.0 PL=0
MOVL C00561 V=800.0 PL=0
MOVL C00562 V=800.0 PL=0
MOVL C00563 V=800.0 PL=0
MOVL C00564 V=800.0 PL=0
MOVL C00565 V=800.0 PL=0
MOVL C00566 V=800.0 PL=0
MOVL C00567 V=800.0 PL=0
MOVL C00568 V=800.0 PL=0
MOVL C00569 V=800.0 PL=0
MOVL C00570 V=800.0 PL=0
MOVL C00571 V=800.0 PL=0
MOVL C00572 V=800.0 PL=0
MOVL C00573 V=800.0 PL=0
MOVL C00574 V=800.0 PL=0
MOVL C00575 V=800.0 PL=0
MOVL C00576 V=800.0 PL=0
MOVL C00577 V=800.0 PL=0
MOVL C00578 V=800.0 PL=0
MOVL C00579 V=800.0 PL=0
MOVL C00580 V=800.0 PL=0
MOVL C00581 V=800.0 PL=0
MOVL C00582 V=800.0 PL=0
MOVL C00583 V=800.0 PL=0
MOVL C00584 V=800.0 PL=0
MOVL C00585 V=800.0 PL=0
MOVL C00586 V=800.0 PL=0
MOVL C00587 V=800.0 PL=0
MOVL C00588 V=800.0 PL=0
MOVL C00589 V=800.0 PL=0
MOVL C00590 V=800.0 PL=0
MOVL C00591 V=800.0 PL=0
MOVL C00592 V=800.0 PL=0
MOVL C00593 V=800.0 PL=0
MOVL C00594 V=800.0 PL=0
MOVL C00595 V=800.0 PL=0
MOVL C00596 V=800.0 PL=0
MOVL C00597 V=800.0 PL=0
MOVL C00598 V=800.0 PL=0
MOVL C00599 V=800.0 PL=0
MOVL C00600 V=800.0 PL=0
MOVL C00601 V=800.0 PL=0
MOVL C00602 V=800.0 PL=0
MOVL C00603 V=800.0 PL=0
MOVL C00604 V=800.0 PL=0
MOVL C00605 V=800.0 PL=0
MOVL C00606 V=800.0 PL=0
MOVL C00607 V=800.0 PL=0
MOVL C00608 V=800.0 PL=0
MOVL C00609 V=800.0 PL=0
MOVL C00610 V=800.0 PL=0
MOVL C00611 V=800.0 PL=0
MOVL C00612 V=800.0 PL=0
MOVL C00613 V=800.0 PL=0
MOVL C00614 V=800.0 PL=0
MOVL C00615 V=800.0 PL=0
MOVL C00616 V=800.0 PL=0
MOVL C00617 V=800.0 PL=0
MOVL C00618 V=800.0 PL=0
MOVL C00619 V=800.0 PL=0
MOVL C00620 V=800.0 PL=0
MOVL C00621 V=800.0 PL=0
MOVL C00622 V=800.0 PL=0
MOVL C00623 V=800.0 PL=0
MOVL C00624 V=800.0 PL=0
MOVL C00625 V=800.0 PL=0
MOVL C00626 V=800.0 PL=0
MOVL C00627 V=800.0 PL=0
MOVL C00628 V=800.0 PL=0
MOVL C00629 V=800.0 PL=0
MOVL C00630 V=800.0 PL=0
MOVL C00631 V=800.0 PL=0
MOVL C00632 V=800.0 PL=0
MOVL C00633 V=800.0 PL=0
MOVL C00634 V=800.0 PL=0
MOVL C00635 V=800.0 PL=0
MOVL C00636 V=800.0 PL=0
MOVL C00637 V=800.0 PL=0
MOVL C00638 V=800.0 PL=0
MOVL C00639 V=800.0 PL=0
MOVL C00640 V=800.0 PL=0
MOVL C00641 V=800.0 PL=0
MOVL C00642 V=800.0 PL=0
MOVL C00643 V=800.0 PL=0
MOVL C00644 V=800.0 PL=0
MOVL C00645 V=800.0 PL=0
MOVL C00646 V=800.0 PL=0
MOVL C00647 V=800.0 PL=0
MOVL C00648 V=800.0 PL=0
MOVL C00649 V=800.0 PL=0
MOVL C00650 V=800.0 PL=0
MOVL C00651 V=800.0 PL=0
MOVL C00652 V=800.0 PL=0
MOVL C00653 V=800.0 PL=0
MOVL C00654 V=800.0 PL=0
MOVL C00655 V=800.0 PL=0
MOVL C00656 V=800.0 PL=0
MOVL C00657 V=800.0 PL=0
MOVL C00658 V=800.0 PL=0
MOVL C00659 V=800.0 PL=0
MOVL C00660 V=800.0 PL=0
MOVL C00661 V=800.0 PL=0
MOVL C00662 V=800.0 PL=0
MOVL C00663 V=800.0 PL=0
MOVL C00664 V=800.0 PL=0
MOVL C00665 V=800.0 PL=0
MOVL C00666 V=800.0 PL=0
MOVL C00667 V=800.0 PL=0
MOVL C00668 V=800.0 PL=0
MOVL C00669 V=800.0 PL=0
MOVL C00670 V=800.0 PL=0
MOVL C00671 V=800.0 PL=0
MOVL C00672 V=800.0 PL=0
MOVL C00673 V=800.0 PL=0
MOVL C00674 V=800.0 PL=0
MOVL C00675 V=800.0 PL=0
MOVL C00676 V=800.0 PL=0
MOVL C00677 V=800.0 PL=0
MOVL C00678 V=800.0 PL=0
MOVL C00679 V=800.0 PL=0
MOVL C00680 V=800.0 PL=0
MOVL C00681 V=800.0 PL=0
MOVL C00682 V=800.0 PL=0
MOVL C00683 V=800.0 PL=0
MOVL C00684 V=800.0 PL=0
MOVL C00685 V=800.0 PL=0
MOVL C00686 V=800.0 PL=0
MOVL C00687 V=800.0 PL=0
MOVL C00688 V=800.0 PL=0
MOVL C00689 V=800.0 PL=0
MOVL C00690 V=800.0 PL=0
MOVL C00691 V=800.0 PL=0
MOVL C00692 V=800.0 PL=0
MOVL C00693 V=800.0 PL=0
MOVL C00694 V=800.0 PL=0
MOVL C00695 V=800.0 PL=0
MOVL C00696 V=800.0 PL=0
MOVL C00697 V=800.0 PL=0
MOVL C00698 V=800.0 PL=0
MOVL C00699 V=800.0 PL=0
MOVL C00700 V=800.0 PL=0
MOVL C00701 V=800.0 PL=0
MOVL C00702 V=800.0 PL=0
MOVL C00703 V=800.0 PL=0
MOVL C00704 V=800.0 PL=0
MOVL C00705 V=800.0 PL=0
MOVL C00706 V=800.0 PL=0
MOVL C00707 V=800.0 PL=0
MOVL C00708 V=800.0 PL=0
MOVL C00709 V=800.0 PL=0
MOVL C00710 V=800.0 PL=0
MOVL C00711 V=800.0 PL=0
MOVL C00712 V=800.0 PL=0
MOVL C00713 V=800.0 PL=0
MOVL C00714 V=800.0 PL=0
MOVL C00715 V=800.0 PL=0
MOVL C00716 V=800.0 PL=0
MOVL C00717 V=800.0 PL=0
MOVL C00718 V=800.0 PL=0
MOVL C00719 V=800.0 PL=0
MOVL C00720 V=800.0 PL=0
MOVL C00721 V=800.0 PL=0
MOVL C00722 V=800.0 PL=0
MOVL C00723 V=800.0 PL=0
MOVL C00724 V=800.0 PL=0
MOVL C00725 V=800.0 PL=0
MOVL C00726 V=800.0 PL=0
MOVL C00727 V=800.0 PL=0
MOVL C00728 V=800.0 PL=0
MOVL C00729 V=800.0 PL=0
MOVL C00730 V=800.0 PL=0
MOVL C00731 V=800.0 PL=0
MOVL C00732 V=800.0 PL=0
MOVL C00733 V=800.0 PL=0
MOVL C00734 V=800.0 PL=0
MOVL C00735 V=800.0 PL=0
MOVL C00736 V=800.0 PL=0
MOVL C00737 V=800.0 PL=0
MOVL C00738 V=800.0 PL=0
MOVL C00739 V=800.0 PL=0
MOVL C00740 V=800.0 PL=0
MOVL C00741 V=800.0 PL=0
MOVL C00742 V=800.0 PL=0
MOVL C00743 V=800.0 PL=0
MOVL C00744 V=800.0 PL=0
MOVL C00745 V=800.0 PL=0
MOVL C00746 V=800.0 PL=0
MOVL C00747 V=800.0 PL=0
MOVL C00748 V=800.0 PL=0
MOVL C00749 V=800.0 PL=0
MOVL C00750 V=800.0 PL=0
MOVL C00751 V=800.0 PL=0
MOVL C00752 V=800.0 PL=0
MOVL C00753 V=800.0 PL=0
MOVL C00754 V=800.0 PL=0
MOVL C00755 V=800.0 PL=0
MOVL C00756 V=800.0 PL=0
MOVL C00757 V=800.0 PL=0
MOVL C00758 V=800.0 PL=0
MOVL C00759 V=800.0 PL=0
MOVL C00760 V=800.0 PL=0
MOVL C00761 V=800.0 PL=0
MOVL C00762 V=800.0 PL=0
MOVL C00763 V=800.0 PL=0
MOVL C00764 V=800.0 PL=0
MOVL C00765 V=800.0 PL=0
MOVL C00766 V=800.0 PL=0
MOVL C00767 V=800.0 PL=0
MOVL C00768 V=800.0 PL=0
MOVL C00769 V=800.0 PL=0
MOVL C00770 V=800.0 PL=0
MOVL C00771 V=800.0 PL=0
MOVL C00772 V=800.0 PL=0
MOVL C00773 V=800.0 PL=0
MOVL C00774 V=800.0 PL=0
MOVL C00775 V=800.0 PL=0
MOVL C00776 V=800.0 PL=0
MOVL C00777 V=800.0 PL=0
MOVL C00778 V=800.0 PL=0
MOVL C00779 V=800.0 PL=0
MOVL C00780 V=800.0 PL=0
MOVL C00781 V=800.0 PL=0
MOVL C00782 V=800.0 PL=0
MOVL C00783 V=800.0 PL=0
MOVL C00784 V=800.0 PL=0
MOVL C00785 V=800.0 PL=0
MOVL C00786 V=800.0 PL=0
MOVL C00787 V=800.0 PL=0
MOVL C00788 V=800.0 PL=0
MOVL C00789 V=800.0 PL=0
MOVL C00790 V=800.0 PL=0
MOVL C00791 V=800.0 PL=0
MOVL C00792 V=800.0 PL=0
MOVL C00793 V=800.0 PL=0
MOVL C00794 V=800.0 PL=0
MOVL C00795 V=800.0 PL=0
MOVL C00796 V=800.0 PL=0
MOVL C00797 V=800.0 PL=0
MOVL C00798 V=800.0 PL=0
MOVL C00799 V=800.0 PL=0
MOVL C00800 V=800.0 PL=0
MOVL C00801 V=800.0 PL=0
MOVL C00802 V=800.0 PL=0
MOVL C00803 V=800.0 PL=0
MOVL C00804 V=800.0 PL=0
MOVL C00805 V=800.0 PL=0
MOVL C00806 V=800.0 PL=0
MOVL C00807 V=800.0 PL=0
MOVL C00808 V=800.0 PL=0
MOVL C00809 V=800.0 PL=0
MOVL C00810 V=800.0 PL=0
MOVL C00811 V=800.0 PL=0
MOVL C00812 V=800.0 PL=0
MOVL C00813 V=800.0 PL=0
MOVL C00814 V=800.0 PL=0
MOVL C00815 V=800.0 PL=0
MOVL C00816 V=800.0 PL=0
MOVL C00817 V=800.0 PL=0
MOVL C00818 V=800.0 PL=0
MOVL C00819 V=800.0 PL=0
MOVL C00820 V=800.0 PL=0
MOVL C00821 V=800.0 PL=0
MOVL C00822 V=800.0 PL=0
MOVL C00823 V=800.0 PL=0
MOVL C00824 V=800.0 PL=0
MOVL C00825 V=800.0 PL=0
MOVL C00826 V=800.0 PL=0
MOVL C00827 V=800.0 PL=0
MOVL C00828 V=800.0 PL=0
MOVL C00829 V=800.0 PL=0
MOVL C00830 V=800.0 PL=0
MOVL C00831 V=800.0 PL=0
MOVL C00832 V=800.0 PL=0
MOVL C00833 V=800.0 PL=0
MOVL C00834 V=800.0 PL=0
MOVL C00835 V=800.0 PL=0
MOVL C00836 V=800.0 PL=0
MOVL C00837 V=800.0 PL=0
MOVL C00838 V=800.0 PL=0
MOVL C00839 V=800.0 PL=0
MOVL C00840 V=800.0 PL=0
MOVL C00841 V=800.0 PL=0
MOVL C00842 V=800.0 PL=0
MOVL C00843 V=800.0 PL=0
MOVL C00844 V=800.0 PL=0
MOVL C00845 V=800.0 PL=0
MOVL C00846 V=800.0 PL=0
MOVL C00847 V=800.0 PL=0
MOVL C00848 V=800.0 PL=0
MOVL C00849 V=800.0 PL=0
MOVL C00850 V=800.0 PL=0
MOVL C00851 V=800.0 PL=0
MOVL C00852 V=800.0 PL=0
MOVL C00853 V=800.0 PL=0
MOVL C00854 V=800.0 PL=0
MOVL C00855 V=800.0 PL=0
MOVL C00856 V=800.0 PL=0
MOVL C00857 V=800.0 PL=0
MOVL C00858 V=800.0 PL=0
MOVL C00859 V=800.0 PL=0
MOVL C00860 V=800.0 PL=0
MOVL C00861 V=800.0 PL=0
MOVL C00862 V=800.0 PL=0
MOVL C00863 V=800.0 PL=0
MOVL C00864 V=800.0 PL=0
MOVL C00865 V=800.0 PL=0
MOVL C00866 V=800.0 PL=0
MOVL C00867 V=800.0 PL=0
MOVL C00868 V=800.0 PL=0
MOVL C00869 V=800.0 PL=0
MOVL C00870 V=800.0 PL=0
MOVL C00871 V=800.0 PL=0
MOVL C00872 V=800.0 PL=0
MOVL C00873 V=800.0 PL=0
MOVL C00874 V=800.0 PL=0
MOVL C00875 V=800.0 PL=0
MOVL C00876 V=800.0 PL=0
MOVL C00877 V=800.0 PL=0
MOVL C00878 V=800.0 PL=0
MOVL C00879 V=800.0 PL=0
MOVL C00880 V=800.0 PL=0
MOVL C00881 V=800.0 PL=0
MOVL C00882 V=800.0 PL=0
MOVL C00883 V=800.0 PL=0
MOVL C00884 V=800.0 PL=0
MOVL C00885 V=800.0 PL=0
MOVL C00886 V=800.0 PL=0
MOVL C00887 V=800.0 PL=0
MOVL C00888 V=800.0 PL=0
MOVL C00889 V=800.0 PL=0
MOVL C00890 V=800.0 PL=0
MOVL C00891 V=800.0 PL=0
MOVL C00892 V=800.0 PL=0
MOVL C00893 V=800.0 PL=0
MOVL C00894 V=800.0 PL=0
MOVL C00895 V=800.0 PL=0
MOVL C00896 V=800.0 PL=0
MOVL C00897 V=800.0 PL=0
MOVL C00898 V=800.0 PL=0
MOVL C00899 V=800.0 PL=0
MOVL C00900 V=800.0 PL=0
MOVL C00901 V=800.0 PL=0
MOVL C00902 V=800.0 PL=0
MOVL C00903 V=800.0 PL=0
MOVL C00904 V=800.0 PL=0
MOVL C00905 V=800.0 PL=0
MOVL C00906 V=800.0 PL=0
MOVL C00907 V=800.0 PL=0
MOVL C00908 V=800.0 PL=0
MOVL C00909 V=800.0 PL=0
MOVL C00910 V=800.0 PL=0
MOVL C00911 V=800.0 PL=0
MOVL C00912 V=800.0 PL=0
MOVL C00913 V=800.0 PL=0
MOVL C00914 V=800.0 PL=0
MOVL C00915 V=800.0 PL=0
MOVL C00916 V=800.0 PL=0
MOVL C00917 V=800.0 PL=0
MOVL C00918 V=800.0 PL=0
MOVL C00919 V=800.0 PL=0
MOVL C00920 V=800.0 PL=0
MOVL C00921 V=800.0 PL=0
MOVL C00922 V=800.0 PL=0
MOVL C00923 V=800.0 PL=0
MOVL C00924 V=800.0 PL=0
MOVL C00925 V=800.0 PL=0
MOVL C00926 V=800.0 PL=0
MOVL C00927 V=800.0 PL=0
MOVL C00928 V=800.0 PL=0
MOVL C00929 V=800.0 PL=0
MOVL C00930 V=800.0 PL=0
MOVL C00931 V=800.0 PL=0
MOVL C00932 V=800.0 PL=0
MOVL C00933 V=800.0 PL=0
MOVL C00934 V=800.0 PL=0
MOVL C00935 V=800.0 PL=0
MOVL C00936 V=800.0 PL=0
MOVL C00937 V=800.0 PL=0
MOVL C00938 V=800.0 PL=0
MOVL C00939 V=800.0 PL=0
MOVL C00940 V=800.0 PL=0
MOVL C00941 V=800.0 PL=0
MOVL C00942 V=800.0 PL=0
MOVL C00943 V=800.0 PL=0
MOVL C00944 V=800.0 PL=0
MOVL C00945 V=800.0 PL=0
MOVL C00946 V=800.0 PL=0
MOVL C00947 V=800.0 PL=0
MOVL C00948 V=800.0 PL=0
MOVL C00949 V=800.0 PL=0
MOVL C00950 V=800.0 PL=0
MOVL C00951 V=800.0 PL=0
MOVL C00952 V=800.0 PL=0
MOVL C00953 V=800.0 PL=0
MOVL C00954 V=800.0 PL=0
MOVL C00955 V=800.0 PL=0
MOVL C00956 V=800.0 PL=0
MOVL C00957 V=800.0 PL=0
MOVL C00958 V=800.0 PL=0
MOVL C00959 V=800.0 PL=0
MOVL C00960 V=800.0 PL=0
MOVL C00961 V=800.0 PL=0
MOVL C00962 V=800.0 PL=0
MOVL C00963 V=800.0 PL=0
MOVL C00964 V=800.0 PL=0
MOVL C00965 V=800.0 PL=0
MOVL C00966 V=800.0 PL=0
MOVL C00967 V=800.0 PL=0
MOVL C00968 V=800.0 PL=0
MOVL C00969 V=800.0 PL=0
MOVL C00970 V=800.0 PL=0
MOVL C00971 V=800.0 PL=0
MOVL C00972 V=800.0 PL=0
MOVL C00973 V=800.0 PL=0
MOVL C00974 V=800.0 PL=0
MOVL C00975 V=800.0 PL=0
MOVL C00976 V=800.0 PL=0
MOVL C00977 V=800.0 PL=0
MOVL C00978 V=800.0 PL=0
MOVL C00979 V=800.0 PL=0
MOVL C00980 V=800.0 PL=0
MOVL C00981 V=800.0 PL=0
MOVL C00982 V=800.0 PL=0
MOVL C00983 V=800.0 PL=0
MOVL C00984 V=800.0 PL=0
MOVL C00985 V=800.0 PL=0
MOVL C00986 V=800.0 PL=0
MOVL C00987 V=800.0 PL=0
MOVL C00988 V=800.0 PL=0
MOVL C00989 V=800.0 PL=0
MOVL C00990 V=800.0 PL=0
MOVL C00991 V=800.0 PL=0
MOVL C00992 V=800.0 PL=0
MOVL C00993 V=800.0 PL=0
MOVL C00994 V=800.0 PL=0
MOVL C00995 V=800.0 PL=0
MOVL C00996 V=800.0 PL=0
MOVL C00997 V=800.0 PL=0
MOVL C00998 V=800.0 PL=0
MOVL C00999 V=800.0 PL=0
MOVL C01000 V=800.0 PL=0
MOVL C01001 V=800.0 PL=0
MOVL C01002 V=800.0 PL=0
MOVL C01003 V=800.0 PL=0
MOVL C01004 V=800.0 PL=0
MOVL C01005 V=800.0 PL=0
MOVL C01006 V=800.0 PL=0
MOVL C01007 V=800.0 PL=0
MOVL C01008 V=800.0 PL=0
MOVL C01009 V=800.0 PL=0
MOVL C01010 V=800.0 PL=0
MOVL C01011 V=800.0 PL=0
MOVL C01012 V=800.0 PL=0
MOVL C01013 V=800.0 PL=0
MOVL C01014 V=800.0 PL=0
MOVL C01015 V=800.0 PL=0
MOVL C01016 V=800.0 PL=0
MOVL C01017 V=800.0 PL=0
MOVL C01018 V=800.0 PL=0
MOVL C01019 V=800.0 PL=0
MOVL C01020 V=800.0 PL=0
MOVL C01021 V=800.0 PL=0
MOVL C01022 V=800.0 PL=0
MOVL C01023 V=800.0 PL=0
MOVL C01024 V=800.0 PL=0
MOVL C01025 V=800.0 PL=0
MOVL C01026 V=800.0 PL=0
MOVL C01027 V=800.0 PL=0
MOVL C01028 V=800.0 PL=0
MOVL C01029 V=800.0 PL=0
MOVL C01030 V=800.0 PL=0
MOVL C01031 V=800.0 PL=0
MOVL C01032 V=800.0 PL=0
MOVL C01033 V=800.0 PL=0
MOVL C01034 V=800.0 PL=0
MOVL C01035 V=800.0 PL=0
MOVL C01036 V=800.0 PL=0
MOVL C01037 V=800.0 PL=0
MOVL C01038 V=800.0 PL=0
MOVL C01039 V=800.0 PL=0
MOVL C01040 V=800.0 PL=0
MOVL C01041 V=800.0 PL=0
MOVL C01042 V=800.0 PL=0
MOVL C01043 V=800.0 PL=0
MOVL C01044 V=800.0 PL=0
MOVL C01045 V=800.0 PL=0
MOVL C01046 V=800.0 PL=0
MOVL C01047 V=800.0 PL=0
MOVL C01048 V=800.0 PL=0
MOVL C01049 V=800.0 PL=0
MOVL C01050 V=800.0 PL=0
MOVL C01051 V=800.0 PL=0
MOVL C01052 V=800.0 PL=0
MOVL C01053 V=800.0 PL=0
MOVL C01054 V=800.0 PL=0
MOVL C01055 V=800.0 PL=0
MOVL C01056 V=800.0 PL=0
MOVL C01057 V=800.0 PL=0
MOVL C01058 V=800.0 PL=0
MOVL C01059 V=800.0 PL=0
MOVL C01060 V=800.0 PL=0
MOVL C01061 V=800.0 PL=0
MOVL C01062 V=800.0 PL=0
MOVL C01063 V=800.0 PL=0
MOVL C01064 V=800.0 PL=0
MOVL C01065 V=800.0 PL=0
MOVL C01066 V=800.0 PL=0
MOVL C01067 V=800.0 PL=0
MOVL C01068 V=800.0 PL=0
MOVL C01069 V=800.0 PL=0
MOVL C01070 V=800.0 PL=0
MOVL C01071 V=800.0 PL=0
MOVL C01072 V=800.0 PL=0
MOVL C01073 V=800.0 PL=0
MOVL C01074 V=800.0 PL=0
MOVL C01075 V=800.0 PL=0
MOVL C01076 V=800.0 PL=0
MOVL C01077 V=800.0 PL=0
MOVL C01078 V=800.0 PL=0
MOVL C01079 V=800.0 PL=0
MOVL C01080 V=800.0 PL=0
MOVL C01081 V=800.0 PL=0
MOVL C01082 V=800.0 PL=0
MOVL C01083 V=800.0 PL=0
MOVL C01084 V=800.0 PL=0
MOVL C01085 V=800.0 PL=0
MOVL C01086 V=800.0 PL=0
MOVL C01087 V=800.0 PL=0
MOVL C01088 V=800.0 PL=0
MOVL C01089 V=800.0 PL=0
MOVL C01090 V=800.0 PL=0
MOVL C01091 V=800.0 PL=0
MOVL C01092 V=800.0 PL=0
MOVL C01093 V=800.0 PL=0
MOVL C01094 V=800.0 PL=0
MOVL C01095 V=800.0 PL=0
MOVL C01096 V=800.0 PL=0
MOVL C01097 V=800.0 PL=0
MOVL C01098 V=800.0 PL=0
MOVL C01099 V=800.0 PL=0
MOVL C01100 V=800.0 PL=0
MOVL C01101 V=800.0 PL=0
MOVL C01102 V=800.0 PL=0
MOVL C01103 V=800.0 PL=0
MOVL C01104 V=800.0 PL=0
MOVL C01105 V=800.0 PL=0
MOVL C01106 V=800.0 PL=0
MOVL C01107 V=800.0 PL=0
MOVL C01108 V=800.0 PL=0
MOVL C01109 V=800.0 PL=0
MOVL C01110 V=800.0 PL=0
MOVL C01111 V=800.0 PL=0
MOVL C01112 V=800.0 PL=0
MOVL C01113 V=800.0 PL=0
MOVL C01114 V=800.0 PL=0
MOVL C01115 V=800.0 PL=0
MOVL C01116 V=800.0 PL=0
MOVL C01117 V=800.0 PL=0
MOVL C01118 V=800.0 PL=0
MOVL C01119 V=800.0 PL=0
MOVL C01120 V=800.0 PL=0
MOVL C01121 V=800.0 PL=0
MOVL C01122 V=800.0 PL=0
MOVL C01123 V=800.0 PL=0
MOVL C01124 V=800.0 PL=0
MOVL C01125 V=800.0 PL=0
MOVL C01126 V=800.0 PL=0
MOVL C01127 V=800.0 PL=0
MOVL C01128 V=800.0 PL=0
MOVL C01129 V=800.0 PL=0
MOVL C01130 V=800.0 PL=0
MOVL C01131 V=800.0 PL=0
MOVL C01132 V=800.0 PL=0
MOVL C01133 V=800.0 PL=0
MOVL C01134 V=800.0 PL=0
MOVL C01135 V=800.0 PL=0
MOVL C01136 V=800.0 PL=0
MOVL C01137 V=800.0 PL=0
MOVL C01138 V=800.0 PL=0
MOVL C01139 V=800.0 PL=0
MOVL C01140 V=800.0 PL=0
MOVL C01141 V=800.0 PL=0
MOVL C01142 V=800.0 PL=0
MOVL C01143 V=800.0 PL=0
MOVL C01144 V=800.0 PL=0
MOVL C01145 V=800.0 PL=0
MOVL C01146 V=800.0 PL=0
MOVL C01147 V=800.0 PL=0
MOVL C01148 V=800.0 PL=0
MOVL C01149 V=800.0 PL=0
MOVL C01150 V=800.0 PL=0
MOVL C01151 V=800.0 PL=0
MOVL C01152 V=800.0 PL=0
MOVL C01153 V=800.0 PL=0
MOVL C01154 V=800.0 PL=0
MOVL C01155 V=800.0 PL=0
MOVL C01156 V=800.0 PL=0
MOVL C01157 V=800.0 PL=0
MOVL C01158 V=800.0 PL=0
MOVL C01159 V=800.0 PL=0
MOVL C01160 V=800.0 PL=0
MOVL C01161 V=800.0 PL=0
MOVL C01162 V=800.0 PL=0
MOVL C01163 V=800.0 PL=0
MOVL C01164 V=800.0 PL=0
MOVL C01165 V=800.0 PL=0
MOVL C01166 V=800.0 PL=0
MOVL C01167 V=800.0 PL=0
MOVL C01168 V=800.0 PL=0
MOVL C01169 V=800.0 PL=0
MOVL C01170 V=800.0 PL=0
MOVL C01171 V=800.0 PL=0
MOVL C01172 V=800.0 PL=0
MOVL C01173 V=800.0 PL=0
MOVL C01174 V=800.0 PL=0
MOVL C01175 V=800.0 PL=0
MOVL C01176 V=800.0 PL=0
MOVL C01177 V=800.0 PL=0
MOVL C01178 V=800.0 PL=0
MOVL C01179 V=800.0 PL=0
MOVL C01180 V=800.0 PL=0
MOVL C01181 V=800.0 PL=0
MOVL C01182 V=800.0 PL=0
MOVL C01183 V=800.0 PL=0
MOVL C01184 V=800.0 PL=0
MOVL C01185 V=800.0 PL=0
MOVL C01186 V=800.0 PL=0
MOVL C01187 V=800.0 PL=0
MOVL C01188 V=800.0 PL=0
MOVL C01189 V=800.0 PL=0
MOVL C01190 V=800.0 PL=0
MOVL C01191 V=800.0 PL=0
MOVL C01192 V=800.0 PL=0
MOVL C01193 V=800.0 PL=0
MOVL C01194 V=800.0 PL=0
MOVL C01195 V=800.0 PL=0
MOVL C01196 V=800.0 PL=0
MOVL C01197 V=800.0 PL=0
MOVL C01198 V=800.0 PL=0
MOVL C01199 V=800.0 PL=0
MOVL C01200 V=800.0 PL=0
MOVL C01201 V=800.0 PL=0
MOVL C01202 V=800.0 PL=0
MOVL C01203 V=800.0 PL=0
MOVL C01204 V=800.0 PL=0
MOVL C01205 V=800.0 PL=0
MOVL C01206 V=800.0 PL=0
MOVL C01207 V=800.0 PL=0
MOVL C01208 V=800.0 PL=0
MOVL C01209 V=800.0 PL=0
MOVL C01210 V=800.0 PL=0
MOVL C01211 V=800.0 PL=0
MOVL C01212 V=800.0 PL=0
MOVL C01213 V=800.0 PL=0
MOVL C01214 V=800.0 PL=0
MOVL C01215 V=800.0 PL=0
MOVL C01216 V=800.0 PL=0
MOVL C01217 V=800.0 PL=0
MOVL C01218 V=800.0 PL=0
MOVL C01219 V=800.0 PL=0
MOVL C01220 V=800.0 PL=0
MOVL C01221 V=800.0 PL=0
MOVL C01222 V=800.0 PL=0
MOVL C01223 V=800.0 PL=0
MOVL C01224 V=800.0 PL=0
MOVL C01225 V=800.0 PL=0
MOVL C01226 V=800.0 PL=0
MOVL C01227 V=800.0 PL=0
MOVL C01228 V=800.0 PL=0
MOVL C01229 V=800.0 PL=0
MOVL C01230 V=800.0 PL=0
MOVL C01231 V=800.0 PL=0
MOVL C01232 V=800.0 PL=0
MOVL C01233 V=800.0 PL=0
MOVL C01234 V=800.0 PL=0
MOVL C01235 V=800.0 PL=0
MOVL C01236 V=800.0 PL=0
MOVL C01237 V=800.0 PL=0
MOVL C01238 V=800.0 PL=0
MOVL C01239 V=800.0 PL=0
MOVL C01240 V=800.0 PL=0
MOVL C01241 V=800.0 PL=0
MOVL C01242 V=800.0 PL=0
MOVL C01243 V=800.0 PL=0
MOVL C01244 V=800.0 PL=0
MOVL C01245 V=800.0 PL=0
MOVL C01246 V=800.0 PL=0
MOVL C01247 V=800.0 PL=0
MOVL C01248 V=800.0 PL=0
MOVL C01249 V=800.0 PL=0
MOVL C01250 V=800.0 PL=0
MOVL C01251 V=800.0 PL=0
MOVL C01252 V=800.0 PL=0
MOVL C01253 V=800.0 PL=0
MOVL C01254 V=800.0 PL=0
MOVL C01255 V=800.0 PL=0
MOVL C01256 V=800.0 PL=0
MOVL C01257 V=800.0 PL=0
MOVL C01258 V=800.0 PL=0
MOVL C01259 V=800.0 PL=0
MOVL C01260 V=800.0 PL=0
MOVL C01261 V=800.0 PL=0
MOVL C01262 V=800.0 PL=0
MOVL C01263 V=800.0 PL=0
MOVL C01264 V=800.0 PL=0
MOVL C01265 V=800.0 PL=0
MOVL C01266 V=800.0 PL=0
MOVL C01267 V=800.0 PL=0
MOVL C01268 V=800.0 PL=0
MOVL C01269 V=800.0 PL=0
MOVL C01270 V=800.0 PL=0
MOVL C01271 V=800.0 PL=0
MOVL C01272 V=800.0 PL=0
MOVL C01273 V=800.0 PL=0
MOVL C01274 V=800.0 PL=0
MOVL C01275 V=800.0 PL=0
MOVL C01276 V=800.0 PL=0
MOVL C01277 V=800.0 PL=0
MOVL C01278 V=800.0 PL=0
MOVL C01279 V=800.0 PL=0
MOVL C01280 V=800.0 PL=0
MOVL C01281 V=800.0 PL=0
MOVL C01282 V=800.0 PL=0
MOVL C01283 V=800.0 PL=0
MOVL C01284 V=800.0 PL=0
MOVL C01285 V=800.0 PL=0
MOVL C01286 V=800.0 PL=0
MOVL C01287 V=800.0 PL=0
MOVL C01288 V=800.0 PL=0
MOVL C01289 V=800.0 PL=0
MOVL C01290 V=800.0 PL=0
MOVL C01291 V=800.0 PL=0
MOVL C01292 V=800.0 PL=0
MOVL C01293 V=800.0 PL=0
MOVL C01294 V=800.0 PL=0
MOVL C01295 V=800.0 PL=0
MOVL C01296 V=800.0 PL=0
MOVL C01297 V=800.0 PL=0
MOVL C01298 V=800.0 PL=0
MOVL C01299 V=800.0 PL=0
MOVL C01300 V=800.0 PL=0
MOVL C01301 V=800.0 PL=0
MOVL C01302 V=800.0 PL=0
MOVL C01303 V=800.0 PL=0
MOVL C01304 V=800.0 PL=0
MOVL C01305 V=800.0 PL=0
MOVL C01306 V=800.0 PL=0
MOVL C01307 V=800.0 PL=0
MOVL C01308 V=800.0 PL=0
MOVL C01309 V=800.0 PL=0
MOVL C01310 V=800.0 PL=0
MOVL C01311 V=800.0 PL=0
MOVL C01312 V=800.0 PL=0
MOVL C01313 V=800.0 PL=0
MOVL C01314 V=800.0 PL=0
MOVL C01315 V=800.0 PL=0
MOVL C01316 V=800.0 PL=0
MOVL C01317 V=800.0 PL=0
MOVL C01318 V=800.0 PL=0
MOVL C01319 V=800.0 PL=0
MOVL C01320 V=800.0 PL=0
MOVL C01321 V=800.0 PL=0
MOVL C01322 V=800.0 PL=0
MOVL C01323 V=800.0 PL=0
MOVL C01324 V=800.0 PL=0
MOVL C01325 V=800.0 PL=0
MOVL C01326 V=800.0 PL=0
MOVL C01327 V=800.0 PL=0
MOVL C01328 V=800.0 PL=0
MOVL C01329 V=800.0 PL=0
MOVL C01330 V=800.0 PL=0
MOVL C01331 V=800.0 PL=0
MOVL C01332 V=800.0 PL=0
MOVL C01333 V=800.0 PL=0
MOVL C01334 V=800.0 PL=0
MOVL C01335 V=800.0 PL=0
MOVL C01336 V=800.0 PL=0
MOVL C01337 V=800.0 PL=0
MOVL C01338 V=800.0 PL=0
MOVL C01339 V=800.0 PL=0
MOVL C01340 V=800.0 PL=0
MOVL C01341 V=800.0 PL=0
MOVL C01342 V=800.0 PL=0
MOVL C01343 V=800.0 PL=0
MOVL C01344 V=800.0 PL=0
MOVL C01345 V=800.0 PL=0
MOVL C01346 V=800.0 PL=0
MOVL C01347 V=800.0 PL=0
MOVL C01348 V=800.0 PL=0
MOVL C01349 V=800.0 PL=0
MOVL C01350 V=800.0 PL=0
MOVL C01351 V=800.0 PL=0
MOVL C01352 V=800.0 PL=0
MOVL C01353 V=800.0 PL=0
MOVL C01354 V=800.0 PL=0
MOVL C01355 V=800.0 PL=0
MOVL C01356 V=800.0 PL=0
MOVL C01357 V=800.0 PL=0
MOVL C01358 V=800.0 PL=0
MOVL C01359 V=800.0 PL=0
MOVL C01360 V=800.0 PL=0
MOVL C01361 V=800.0 PL=0
MOVL C01362 V=800.0 PL=0
MOVL C01363 V=800.0 PL=0
MOVL C01364 V=800.0 PL=0
MOVL C01365 V=800.0 PL=0
MOVL C01366 V=800.0 PL=0
MOVL C01367 V=800.0 PL=0
MOVL C01368 V=800.0 PL=0
MOVL C01369 V=800.0 PL=0
MOVL C01370 V=800.0 PL=0
MOVL C01371 V=800.0 PL=0
MOVL C01372 V=800.0 PL=0
MOVL C01373 V=800.0 PL=0
MOVL C01374 V=800.0 PL=0
MOVL C01375 V=800.0 PL=0
MOVL C01376 V=800.0 PL=0
MOVL C01377 V=800.0 PL=0
MOVL C01378 V=800.0 PL=0
MOVL C01379 V=800.0 PL=0
MOVL C01380 V=800.0 PL=0
MOVL C01381 V=800.0 PL=0
MOVL C01382 V=800.0 PL=0
MOVL C01383 V=800.0 PL=0
MOVL C01384 V=800.0 PL=0
MOVL C01385 V=800.0 PL=0
MOVL C01386 V=800.0 PL=0
MOVL C01387 V=800.0 PL=0
MOVL C01388 V=800.0 PL=0
MOVL C01389 V=800.0 PL=0
MOVL C01390 V=800.0 PL=0
MOVL C01391 V=800.0 PL=0
MOVL C01392 V=800.0 PL=0
MOVL C01393 V=800.0 PL=0
MOVL C01394 V=800.0 PL=0
MOVL C01395 V=800.0 PL=0
MOVL C01396 V=800.0 PL=0
MOVL C01397 V=800.0 PL=0
MOVL C01398 V=800.0 PL=0
MOVL C01399 V=800.0 PL=0
MOVL C01400 V=800.0 PL=0
MOVL C01401 V=800.0 PL=0
MOVL C01402 V=800.0 PL=0
MOVL C01403 V=800.0 PL=0
MOVL C01404 V=800.0 PL=0
MOVL C01405 V=800.0 PL=0
MOVL C01406 V=800.0 PL=0
MOVL C01407 V=800.0 PL=0
MOVL C01408 V=800.0 PL=0
MOVL C01409 V=800.0 PL=0
MOVL C01410 V=800.0 PL=0
MOVL C01411 V=800.0 PL=0
MOVL C01412 V=800.0 PL=0
MOVL C01413 V=800.0 PL=0
MOVL C01414 V=800.0 PL=0
MOVL C01415 V=800.0 PL=0
MOVL C01416 V=800.0 PL=0
MOVL C01417 V=800.0 PL=0
MOVL C01418 V=800.0 PL=0
MOVL C01419 V=800.0 PL=0
MOVL C01420 V=800.0 PL=0
MOVL C01421 V=800.0 PL=0
MOVL C01422 V=800.0 PL=0
MOVL C01423 V=800.0 PL=0
MOVL C01424 V=800.0 PL=0
MOVL C01425 V=800.0 PL=0
MOVL C01426 V=800.0 PL=0
MOVL C01427 V=800.0 PL=0
MOVL C01428 V=800.0 PL=0
MOVL C01429 V=800.0 PL=0
MOVL C01430 V=800.0 PL=0
MOVL C01431 V=800.0 PL=0
MOVL C01432 V=800.0 PL=0
MOVL C01433 V=800.0 PL=0
MOVL C01434 V=800.0 PL=0
MOVL C01435 V=800.0 PL=0
MOVL C01436 V=800.0 PL=0
MOVL C01437 V=800.0 PL=0
MOVL C01438 V=800.0 PL=0
MOVL C01439 V=800.0 PL=0
MOVL C01440 V=800.0 PL=0
MOVL C01441 V=800.0 PL=0
MOVL C01442 V=800.0 PL=0
MOVL C01443 V=800.0 PL=0
MOVL C01444 V=800.0 PL=0
MOVL C01445 V=800.0 PL=0
MOVL C01446 V=800.0 PL=0
MOVL C01447 V=800.0 PL=0
MOVL C01448 V=800.0 PL=0
MOVL C01449 V=800.0 PL=0
MOVL C01450 V=800.0 PL=0
MOVL C01451 V=800.0 PL=0
MOVL C01452 V=800.0 PL=0
MOVL C01453 V=800.0 PL=0
MOVL C01454 V=800.0 PL=0
MOVL C01455 V=800.0 PL=0
MOVL C01456 V=800.0 PL=0
MOVL C01457 V=800.0 PL=0
MOVL C01458 V=800.0 PL=0
MOVL C01459 V=800.0 PL=0
MOVL C01460 V=800.0 PL=0
MOVL C01461 V=800.0 PL=0
MOVL C01462 V=800.0 PL=0
MOVL C01463 V=800.0 PL=0
MOVL C01464 V=800.0 PL=0
MOVL C01465 V=800.0 PL=0
MOVL C01466 V=800.0 PL=0
MOVL C01467 V=800.0 PL=0
MOVL C01468 V=800.0 PL=0
MOVL C01469 V=800.0 PL=0
MOVL C01470 V=800.0 PL=0
MOVL C01471 V=800.0 PL=0
MOVL C01472 V=800.0 PL=0
MOVL C01473 V=800.0 PL=0
MOVL C01474 V=800.0 PL=0
MOVL C01475 V=800.0 PL=0
MOVL C01476 V=800.0 PL=0
MOVL C01477 V=800.0 PL=0
MOVL C01478 V=800.0 PL=0
MOVL C01479 V=800.0 PL=0
MOVL C01480 V=800.0 PL=0
MOVL C01481 V=800.0 PL=0
MOVL C01482 V=800.0 PL=0
MOVL C01483 V=800.0 PL=0
MOVL C01484 V=800.0 PL=0
MOVL C01485 V=800.0 PL=0
MOVL C01486 V=800.0 PL=0
MOVL C01487 V=800.0 PL=0
MOVL C01488 V=800.0 PL=0
MOVL C01489 V=800.0 PL=0
MOVL C01490 V=800.0 PL=0
MOVL C01491 V=800.0 PL=0
MOVL C01492 V=800.0 PL=0
MOVL C01493 V=800.0 PL=0
MOVL C01494 V=800.0 PL=0
MOVL C01495 V=800.0 PL=0
MOVL C01496 V=800.0 PL=0
MOVL C01497 V=800.0 PL=0
MOVL C01498 V=800.0 PL=0
MOVL C01499 V=800.0 PL=0
MOVL C01500 V=800.0 PL=0
MOVL C01501 V=800.0 PL=0
MOVL C01502 V=800.0 PL=0
MOVL C01503 V=800.0 PL=0
MOVL C01504 V=800.0 PL=0
MOVL C01505 V=800.0 PL=0
MOVL C01506 V=800.0 PL=0
MOVL C01507 V=800.0 PL=0
MOVL C01508 V=800.0 PL=0
MOVL C01509 V=800.0 PL=0
MOVL C01510 V=800.0 PL=0
MOVL C01511 V=800.0 PL=0
MOVL C01512 V=800.0 PL=0
MOVL C01513 V=800.0 PL=0
MOVL C01514 V=800.0 PL=0
MOVL C01515 V=800.0 PL=0
MOVL C01516 V=800.0 PL=0
MOVL C01517 V=800.0 PL=0
MOVL C01518 V=800.0 PL=0
MOVL C01519 V=800.0 PL=0
MOVL C01520 V=800.0 PL=0
MOVL C01521 V=800.0 PL=0
MOVL C01522 V=800.0 PL=0
MOVL C01523 V=800.0 PL=0
MOVL C01524 V=800.0 PL=0
MOVL C01525 V=800.0 PL=0
MOVL C01526 V=800.0 PL=0
MOVL C01527 V=800.0 PL=0
MOVL C01528 V=800.0 PL=0
MOVL C01529 V=800.0 PL=0
MOVL C01530 V=800.0 PL=0
MOVL C01531 V=800.0 PL=0
MOVL C01532 V=800.0 PL=0
MOVL C01533 V=800.0 PL=0
MOVL C01534 V=800.0 PL=0
MOVL C01535 V=800.0 PL=0
MOVL C01536 V=800.0 PL=0
MOVL C01537 V=800.0 PL=0
MOVL C01538 V=800.0 PL=0
MOVL C01539 V=800.0 PL=0
MOVL C01540 V=800.0 PL=0
MOVL C01541 V=800.0 PL=0
MOVL C01542 V=800.0 PL=0
MOVL C01543 V=800.0 PL=0
MOVL C01544 V=800.0 PL=0
MOVL C01545 V=800.0 PL=0
MOVL C01546 V=800.0 PL=0
MOVL C01547 V=800.0 PL=0
MOVL C01548 V=800.0 PL=0
MOVL C01549 V=800.0 PL=0
MOVL C01550 V=800.0 PL=0
MOVL C01551 V=800.0 PL=0
MOVL C01552 V=800.0 PL=0
MOVL C01553 V=800.0 PL=0
MOVL C01554 V=800.0 PL=0
MOVL C01555 V=800.0 PL=0
MOVL C01556 V=800.0 PL=0
MOVL C01557 V=800.0 PL=0
MOVL C01558 V=800.0 PL=0
MOVL C01559 V=800.0 PL=0
MOVL C01560 V=800.0 PL=0
MOVL C01561 V=800.0 PL=0
MOVL C01562 V=800.0 PL=0
MOVL C01563 V=800.0 PL=0
MOVL C01564 V=800.0 PL=0
MOVL C01565 V=800.0 PL=0
MOVL C01566 V=800.0 PL=0
MOVL C01567 V=800.0 PL=0
MOVL C01568 V=800.0 PL=0
MOVL C01569 V=800.0 PL=0
MOVL C01570 V=800.0 PL=0
MOVL C01571 V=800.0 PL=0
MOVL C01572 V=800.0 PL=0
MOVL C01573 V=800.0 PL=0
MOVL C01574 V=800.0 PL=0
MOVL C01575 V=800.0 PL=0
MOVL C01576 V=800.0 PL=0
MOVL C01577 V=800.0 PL=0
MOVL C01578 V=800.0 PL=0
MOVL C01579 V=800.0 PL=0
MOVL C01580 V=800.0 PL=0
MOVL C01581 V=800.0 PL=0
MOVL C01582 V=800.0 PL=0
MOVL C01583 V=800.0 PL=0
MOVL C01584 V=800.0 PL=0
MOVL C01585 V=800.0 PL=0
MOVL C01586 V=800.0 PL=0
MOVL C01587 V=800.0 PL=0
MOVL C01588 V=800.0 PL=0
MOVL C01589 V=800.0 PL=0
MOVL C01590 V=800.0 PL=0
MOVL C01591 V=800.0 PL=0
MOVL C01592 V=800.0 PL=0
MOVL C01593 V=800.0 PL=0
MOVL C01594 V=800.0 PL=0
MOVL C01595 V=800.0 PL=0
MOVL C01596 V=800.0 PL=0
MOVL C01597 V=800.0 PL=0
MOVL C01598 V=800.0 PL=0
MOVL C01599 V=800.0 PL=0
MOVL C01600 V=800.0 PL=0
MOVL C01601 V=800.0 PL=0
MOVL C01602 V=800.0 PL=0
MOVL C01603 V=800.0 PL=0
MOVL C01604 V=800.0 PL=0
MOVL C01605 V=800.0 PL=0
MOVL C01606 V=800.0 PL=0
MOVL C01607 V=800.0 PL=0
MOVL C01608 V=800.0 PL=0
MOVL C01609 V=800.0 PL=0
MOVL C01610 V=800.0 PL=0
MOVL C01611 V=800.0 PL=0
MOVL C01612 V=800.0 PL=0
MOVL C01613 V=800.0 PL=0
MOVL C01614 V=800.0 PL=0
MOVL C01615 V=800.0 PL=0
MOVL C01616 V=800.0 PL=0
MOVL C01617 V=800.0 PL=0
MOVL C01618 V=800.0 PL=0
MOVL C01619 V=800.0 PL=0
MOVL C01620 V=800.0 PL=0
MOVL C01621 V=800.0 PL=0
MOVL C01622 V=800.0 PL=0
MOVL C01623 V=800.0 PL=0
MOVL C01624 V=800.0 PL=0
MOVL C01625 V=800.0 PL=0
MOVL C01626 V=800.0 PL=0
MOVL C01627 V=800.0 PL=0
MOVL C01628 V=800.0 PL=0
MOVL C01629 V=800.0 PL=0
MOVL C01630 V=800.0 PL=0
MOVL C01631 V=800.0 PL=0
MOVL C01632 V=800.0 PL=0
MOVL C01633 V=800.0 PL=0
MOVL C01634 V=800.0 PL=0
MOVL C01635 V=800.0 PL=0
MOVL C01636 V=800.0 PL=0
MOVL C01637 V=800.0 PL=0
MOVL C01638 V=800.0 PL=0
MOVL C01639 V=800.0 PL=0
MOVL C01640 V=800.0 PL=0
MOVL C01641 V=800.0 PL=0
MOVL C01642 V=800.0 PL=0
MOVL C01643 V=800.0 PL=0
MOVL C01644 V=800.0 PL=0
MOVL C01645 V=800.0 PL=0
MOVL C01646 V=800.0 PL=0
MOVL C01647 V=800.0 PL=0
MOVL C01648 V=800.0 PL=0
MOVL C01649 V=800.0 PL=0
MOVL C01650 V=800.0 PL=0
MOVL C01651 V=800.0 PL=0
MOVL C01652 V=800.0 PL=0
MOVL C01653 V=800.0 PL=0
MOVL C01654 V=800.0 PL=0
MOVL C01655 V=800.0 PL=0
MOVL C01656 V=800.0 PL=0
MOVL C01657 V=800.0 PL=0
MOVL C01658 V=800.0 PL=0
MOVL C01659 V=800.0 PL=0
MOVL C01660 V=800.0 PL=0
MOVL C01661 V=800.0 PL=0
MOVL C01662 V=800.0 PL=0
MOVL C01663 V=800.0 PL=0
MOVL C01664 V=800.0 PL=0
MOVL C01665 V=800.0 PL=0
MOVL C01666 V=800.0 PL=0
MOVL C01667 V=800.0 PL=0
MOVL C01668 V=800.0 PL=0
MOVL C01669 V=800.0 PL=0
MOVL C01670 V=800.0 PL=0
MOVL C01671 V=800.0 PL=0
MOVL C01672 V=800.0 PL=0
MOVL C01673 V=800.0 PL=0
MOVL C01674 V=800.0 PL=0
MOVL C01675 V=800.0 PL=0
MOVL C01676 V=800.0 PL=0
MOVL C01677 V=800.0 PL=0
MOVL C01678 V=800.0 PL=0
MOVL C01679 V=800.0 PL=0
MOVL C01680 V=800.0 PL=0
MOVL C01681 V=800.0 PL=0
MOVL C01682 V=800.0 PL=0
MOVL C01683 V=800.0 PL=0
MOVL C01684 V=800.0 PL=0
MOVL C01685 V=800.0 PL=0
MOVL C01686 V=800.0 PL=0
MOVL C01687 V=800.0 PL=0
MOVL C01688 V=800.0 PL=0
MOVL C01689 V=800.0 PL=0
MOVL C01690 V=800.0 PL=0
MOVL C01691 V=800.0 PL=0
MOVL C01692 V=800.0 PL=0
MOVL C01693 V=800.0 PL=0
MOVL C01694 V=800.0 PL=0
MOVL C01695 V=800.0 PL=0
MOVL C01696 V=800.0 PL=0
MOVL C01697 V=800.0 PL=0
MOVL C01698 V=800.0 PL=0
MOVL C01699 V=800.0 PL=0
MOVL C01700 V=800.0 PL=0
MOVL C01701 V=800.0 PL=0
MOVL C01702 V=800.0 PL=0
MOVL C01703 V=800.0 PL=0
MOVL C01704 V=800.0 PL=0
MOVL C01705 V=800.0 PL=0
MOVL C01706 V=800.0 PL=0
MOVL C01707 V=800.0 PL=0
MOVL C01708 V=800.0 PL=0
MOVL C01709 V=800.0 PL=0
MOVL C01710 V=800.0 PL=0
MOVL C01711 V=800.0 PL=0
MOVL C01712 V=800.0 PL=0
MOVL C01713 V=800.0 PL=0
MOVL C01714 V=800.0 PL=0
MOVL C01715 V=800.0 PL=0
MOVL C01716 V=800.0 PL=0
MOVL C01717 V=800.0 PL=0
MOVL C01718 V=800.0 PL=0
MOVL C01719 V=800.0 PL=0
MOVL C01720 V=800.0 PL=0
MOVL C01721 V=800.0 PL=0
MOVL C01722 V=800.0 PL=0
MOVL C01723 V=800.0 PL=0
MOVL C01724 V=800.0 PL=0
MOVL C01725 V=800.0 PL=0
MOVL C01726 V=800.0 PL=0
MOVL C01727 V=800.0 PL=0
MOVL C01728 V=800.0 PL=0
MOVL C01729 V=800.0 PL=0
MOVL C01730 V=800.0 PL=0
MOVL C01731 V=800.0 PL=0
MOVL C01732 V=800.0 PL=0
MOVL C01733 V=800.0 PL=0
MOVL C01734 V=800.0 PL=0
MOVL C01735 V=800.0 PL=0
MOVL C01736 V=800.0 PL=0
MOVL C01737 V=800.0 PL=0
